Yaskawa INFORM job: vendrediTRJ2.JBI

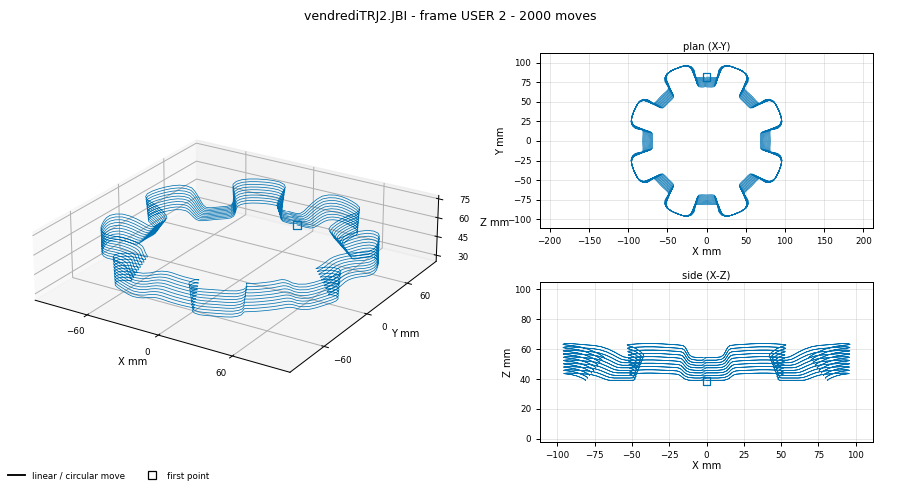
[picture p0: tool path of vendrediTRJ2.JBI in frame USER 2, 2000 of 2000 moves have a stored position in this frame; points joined in program order, loops and branches not executed]
/JOB
//NAME temp/vendrediTRJ2
///FOLDERNAME DEMO
//POS
///NPOS 2000,0,2000,0,0,0
///USER 2
///TOOL 7
///POSTYPE USER
///RECTAN
///RCONF 1,0,0,0,0,0,0,0,0,0,0,0,0,0,0,0,0,0,0,0,0,0,0,0
C00000=0.000,81.307,38.958,180.0000,38.2428,-7290.0000
C00001=4.084,81.202,38.949,-179.8245,38.2510,-7292.8792
C00002=8.115,80.931,38.962,177.3778,38.0004,-7295.7259
C00003=12.050,80.963,39.253,165.4097,32.4399,-7298.4654
C00004=14.402,82.041,39.987,165.7021,8.6017,-7299.9566
C00005=15.932,84.113,41.004,175.9998,1.1820,-7300.7254
C00006=17.234,86.943,42.060,-178.2328,-0.3684,-7301.2119
C00007=18.580,90.119,42.880,-175.4141,-1.1362,-7301.6495
C00008=20.259,92.987,43.289,-175.9026,-2.4170,-7302.2909
C00009=23.317,94.913,43.506,-178.5099,-2.2669,-7303.8024
C00010=27.389,95.566,43.684,-179.5720,-1.5763,-7305.9922
C00011=31.762,94.755,43.864,-179.9981,-0.0779,-7308.5312
C00012=36.110,93.244,43.984,179.9988,-0.0128,-7311.1696
C00013=40.400,91.468,43.984,179.9994,-0.0128,-7313.8303
C00014=44.543,89.461,43.864,179.9999,-0.0769,-7316.4689
C00015=48.209,86.942,43.684,179.5695,-1.5754,-7319.0082
C00016=50.626,83.601,43.506,178.5085,-2.2635,-7321.1977
C00017=51.426,80.077,43.289,175.9070,-2.4130,-7322.7089
C00018=50.586,76.861,42.880,175.4171,-1.1367,-7323.3509
C00019=49.291,73.664,42.060,178.2332,-0.3687,-7323.7878
C00020=48.211,70.742,41.004,-176.0002,1.1799,-7324.2746
C00021=47.828,68.195,39.987,-165.7028,8.5989,-7325.0436
C00022=48.729,65.770,39.253,-165.4121,32.4425,-7326.5348
C00023=51.488,62.965,38.962,-177.3793,38.0014,-7329.2737
C00024=54.531,60.307,38.949,179.8287,38.2519,-7332.1206
C00025=57.493,57.493,38.958,-180.0000,38.2429,-7335.0000
C00026=60.306,54.531,38.949,-179.8283,38.2519,-7337.8789
C00027=62.965,51.488,38.962,177.3793,38.0014,-7340.7263
C00028=65.770,48.729,39.253,165.4121,32.4425,-7343.4652
C00029=68.195,47.828,39.987,165.7028,8.5989,-7344.9564
C00030=70.742,48.211,41.004,176.0002,1.1799,-7345.7254
C00031=73.664,49.291,42.060,-178.2332,-0.3687,-7346.2122
C00032=76.861,50.586,42.880,-175.4171,-1.1367,-7346.6491
C00033=80.077,51.426,43.289,-175.9070,-2.4130,-7347.2911
C00034=83.601,50.626,43.506,-178.5085,-2.2635,-7348.8023
C00035=86.942,48.209,43.684,-179.5695,-1.5754,-7350.9918
C00036=89.461,44.543,43.864,-179.9999,-0.0769,-7353.5311
C00037=91.468,40.400,43.984,-179.9994,-0.0128,-7356.1697
C00038=93.244,36.110,43.984,-179.9988,-0.0128,-7358.8304
C00039=94.755,31.762,43.864,179.9981,-0.0779,-7361.4688
C00040=95.566,27.389,43.684,179.5720,-1.5763,-7364.0078
C00041=94.913,23.317,43.506,178.5099,-2.2669,-7366.1976
C00042=92.987,20.259,43.289,175.9026,-2.4170,-7367.7091
C00043=90.119,18.580,42.880,175.4141,-1.1362,-7368.3505
C00044=86.943,17.234,42.060,178.2328,-0.3684,-7368.7881
C00045=84.113,15.932,41.004,-175.9998,1.1820,-7369.2746
C00046=82.041,14.402,39.987,-165.7021,8.6017,-7370.0434
C00047=80.963,12.050,39.253,-165.4097,32.4399,-7371.5346
C00048=80.931,8.115,38.962,-177.3778,38.0004,-7374.2741
C00049=81.202,4.084,38.949,179.8245,38.2510,-7377.1208
C00050=81.307,0.000,38.958,-180.0000,38.2428,-7380.0000
C00051=81.202,-4.084,38.949,-179.8245,38.2510,-7382.8792
C00052=80.931,-8.116,38.962,177.3773,38.0004,-7385.7266
C00053=80.963,-12.050,39.253,165.4097,32.4399,-7388.4654
C00054=82.041,-14.402,39.987,165.7021,8.6017,-7389.9566
C00055=84.113,-15.932,41.004,175.9998,1.1820,-7390.7254
C00056=86.943,-17.234,42.060,-178.2328,-0.3684,-7391.2119
C00057=90.119,-18.580,42.880,-175.4141,-1.1362,-7391.6495
C00058=92.987,-20.259,43.289,-175.9026,-2.4170,-7392.2909
C00059=94.913,-23.317,43.506,-178.5099,-2.2669,-7393.8024
C00060=95.566,-27.389,43.684,-179.5720,-1.5763,-7395.9922
C00061=94.755,-31.762,43.864,-179.9981,-0.0779,-7398.5312
C00062=93.244,-36.110,43.984,179.9988,-0.0128,-7401.1696
C00063=91.468,-40.400,43.984,179.9994,-0.0128,-7403.8303
C00064=89.461,-44.543,43.864,179.9999,-0.0769,-7406.4689
C00065=86.942,-48.209,43.684,179.5695,-1.5754,-7409.0082
C00066=83.601,-50.626,43.506,178.5085,-2.2635,-7411.1977
C00067=80.077,-51.426,43.289,175.9070,-2.4130,-7412.7089
C00068=76.861,-50.586,42.880,175.4171,-1.1367,-7413.3509
C00069=73.664,-49.291,42.060,178.2332,-0.3687,-7413.7878
C00070=70.742,-48.211,41.004,-176.0002,1.1799,-7414.2746
C00071=68.195,-47.828,39.987,-165.7028,8.5989,-7415.0436
C00072=65.770,-48.729,39.253,-165.4121,32.4425,-7416.5348
C00073=62.965,-51.488,38.962,-177.3793,38.0014,-7419.2737
C00074=60.307,-54.531,38.949,179.8287,38.2519,-7422.1206
C00075=57.493,-57.493,38.958,180.0000,38.2429,-7425.0000
C00076=54.531,-60.306,38.949,-179.8283,38.2519,-7427.8789
C00077=51.488,-62.965,38.962,177.3793,38.0014,-7430.7263
C00078=48.729,-65.770,39.253,165.4121,32.4425,-7433.4652
C00079=47.828,-68.195,39.987,165.7028,8.5989,-7434.9564
C00080=48.211,-70.742,41.004,176.0002,1.1799,-7435.7254
C00081=49.291,-73.664,42.060,-178.2332,-0.3687,-7436.2122
C00082=50.586,-76.861,42.880,-175.4171,-1.1367,-7436.6491
C00083=51.426,-80.077,43.289,-175.9070,-2.4130,-7437.2911
C00084=50.626,-83.601,43.506,-178.5085,-2.2635,-7438.8023
C00085=48.209,-86.942,43.684,-179.5695,-1.5754,-7440.9918
C00086=44.543,-89.461,43.864,-179.9999,-0.0769,-7443.5311
C00087=40.400,-91.468,43.984,-179.9994,-0.0128,-7446.1697
C00088=36.110,-93.244,43.984,-179.9988,-0.0128,-7448.8304
C00089=31.762,-94.755,43.864,179.9981,-0.0779,-7451.4688
C00090=27.389,-95.566,43.684,179.5720,-1.5763,-7454.0078
C00091=23.317,-94.913,43.506,178.5099,-2.2669,-7456.1976
C00092=20.259,-92.987,43.289,175.9026,-2.4170,-7457.7091
C00093=18.580,-90.119,42.880,175.4141,-1.1362,-7458.3505
C00094=17.234,-86.943,42.060,178.2328,-0.3684,-7458.7881
C00095=15.932,-84.113,41.004,-175.9998,1.1820,-7459.2746
C00096=14.402,-82.041,39.987,-165.7021,8.6017,-7460.0434
C00097=12.050,-80.963,39.253,-165.4097,32.4399,-7461.5346
C00098=8.115,-80.931,38.962,-177.3778,38.0004,-7464.2741
C00099=4.084,-81.202,38.949,179.8245,38.2510,-7467.1208
C00100=0.000,-81.307,38.958,180.0000,38.2428,-7470.0000
C00101=-4.084,-81.202,38.949,-179.8245,38.2510,-7472.8792
C00102=-8.116,-80.931,38.962,177.3773,38.0004,-7475.7266
C00103=-12.050,-80.963,39.253,165.4097,32.4399,-7478.4654
C00104=-14.402,-82.041,39.987,165.7021,8.6017,-7479.9566
C00105=-15.932,-84.113,41.004,175.9998,1.1820,-7480.7254
C00106=-17.234,-86.943,42.060,-178.2328,-0.3684,-7481.2119
C00107=-18.580,-90.119,42.880,-175.4141,-1.1362,-7481.6495
C00108=-20.259,-92.987,43.289,-175.9026,-2.4170,-7482.2909
C00109=-23.317,-94.913,43.506,-178.5099,-2.2669,-7483.8024
C00110=-27.389,-95.566,43.684,-179.5720,-1.5763,-7485.9922
C00111=-31.762,-94.755,43.864,-179.9981,-0.0779,-7488.5312
C00112=-36.110,-93.244,43.984,179.9988,-0.0128,-7491.1696
C00113=-40.400,-91.468,43.984,179.9994,-0.0128,-7493.8303
C00114=-44.543,-89.461,43.864,179.9999,-0.0769,-7496.4689
C00115=-48.209,-86.942,43.684,179.5695,-1.5754,-7499.0082
C00116=-50.626,-83.601,43.506,178.5085,-2.2635,-7501.1977
C00117=-51.426,-80.077,43.289,175.9070,-2.4130,-7502.7089
C00118=-50.586,-76.861,42.880,175.4171,-1.1367,-7503.3509
C00119=-49.291,-73.664,42.060,178.2332,-0.3687,-7503.7878
C00120=-48.211,-70.742,41.004,-176.0002,1.1799,-7504.2746
C00121=-47.828,-68.195,39.987,-165.7028,8.5989,-7505.0436
C00122=-48.729,-65.770,39.253,-165.4121,32.4425,-7506.5348
C00123=-51.488,-62.965,38.962,-177.3793,38.0014,-7509.2737
C00124=-54.531,-60.307,38.949,179.8287,38.2519,-7512.1206
C00125=-57.493,-57.493,38.958,180.0000,38.2429,-7515.0000
C00126=-60.306,-54.531,38.949,-179.8283,38.2519,-7517.8789
C00127=-62.965,-51.488,38.962,177.3793,38.0014,-7520.7263
C00128=-65.770,-48.729,39.253,165.4121,32.4425,-7523.4652
C00129=-68.195,-47.828,39.987,165.7028,8.5989,-7524.9564
C00130=-70.742,-48.211,41.004,176.0002,1.1799,-7525.7254
C00131=-73.664,-49.291,42.060,-178.2332,-0.3687,-7526.2122
C00132=-76.861,-50.586,42.880,-175.4171,-1.1367,-7526.6491
C00133=-80.077,-51.426,43.289,-175.9070,-2.4130,-7527.2911
C00134=-83.601,-50.626,43.506,-178.5085,-2.2635,-7528.8023
C00135=-86.942,-48.209,43.684,-179.5695,-1.5754,-7530.9918
C00136=-89.461,-44.543,43.864,-179.9999,-0.0769,-7533.5311
C00137=-91.468,-40.400,43.984,-179.9994,-0.0128,-7536.1697
C00138=-93.244,-36.110,43.984,-179.9988,-0.0128,-7538.8304
C00139=-94.755,-31.762,43.864,179.9981,-0.0779,-7541.4688
C00140=-95.566,-27.389,43.684,179.5720,-1.5763,-7544.0078
C00141=-94.913,-23.317,43.506,178.5099,-2.2669,-7546.1976
C00142=-92.987,-20.259,43.289,175.9026,-2.4170,-7547.7091
C00143=-90.119,-18.580,42.880,175.4141,-1.1362,-7548.3505
C00144=-86.943,-17.234,42.060,178.2328,-0.3684,-7548.7881
C00145=-84.113,-15.932,41.004,-175.9998,1.1820,-7549.2746
C00146=-82.041,-14.402,39.987,-165.7021,8.6017,-7550.0434
C00147=-80.963,-12.050,39.253,-165.4097,32.4399,-7551.5346
C00148=-80.931,-8.115,38.962,-177.3778,38.0004,-7554.2741
C00149=-81.202,-4.084,38.949,179.8245,38.2510,-7557.1208
C00150=-81.307,0.000,38.958,180.0000,38.2428,-7560.0000
C00151=-81.202,4.084,38.949,-179.8245,38.2510,-7562.8792
C00152=-80.931,8.116,38.962,177.3773,38.0004,-7565.7266
C00153=-80.963,12.050,39.253,165.4097,32.4399,-7568.4654
C00154=-82.041,14.402,39.987,165.7021,8.6017,-7569.9566
C00155=-84.113,15.932,41.004,175.9998,1.1820,-7570.7254
C00156=-86.943,17.234,42.060,-178.2328,-0.3684,-7571.2119
C00157=-90.119,18.580,42.880,-175.4141,-1.1362,-7571.6495
C00158=-92.987,20.259,43.289,-175.9026,-2.4170,-7572.2909
C00159=-94.913,23.317,43.506,-178.5099,-2.2669,-7573.8024
C00160=-95.566,27.389,43.684,-179.5720,-1.5763,-7575.9922
C00161=-94.755,31.762,43.864,-179.9981,-0.0779,-7578.5312
C00162=-93.244,36.110,43.984,179.9988,-0.0128,-7581.1696
C00163=-91.468,40.400,43.984,179.9994,-0.0128,-7583.8303
C00164=-89.461,44.543,43.864,179.9999,-0.0769,-7586.4689
C00165=-86.942,48.209,43.684,179.5695,-1.5754,-7589.0082
C00166=-83.601,50.626,43.506,178.5085,-2.2635,-7591.1977
C00167=-80.077,51.426,43.289,175.9070,-2.4130,-7592.7089
C00168=-76.861,50.586,42.880,175.4171,-1.1367,-7593.3509
C00169=-73.664,49.291,42.060,178.2332,-0.3687,-7593.7878
C00170=-70.742,48.211,41.004,-176.0002,1.1799,-7594.2746
C00171=-68.195,47.828,39.987,-165.7028,8.5989,-7595.0436
C00172=-65.770,48.729,39.253,-165.4121,32.4425,-7596.5348
C00173=-62.965,51.488,38.962,-177.3793,38.0014,-7599.2737
C00174=-60.307,54.531,38.949,179.8287,38.2519,-7602.1206
C00175=-57.493,57.493,38.958,-180.0000,38.2429,-7605.0000
C00176=-54.531,60.306,38.949,-179.8283,38.2519,-7607.8789
C00177=-51.488,62.965,38.962,177.3793,38.0014,-7610.7263
C00178=-48.729,65.770,39.253,165.4121,32.4425,-7613.4652
C00179=-47.828,68.195,39.987,165.7028,8.5989,-7614.9564
C00180=-48.211,70.742,41.004,176.0002,1.1799,-7615.7254
C00181=-49.291,73.664,42.060,-178.2332,-0.3687,-7616.2122
C00182=-50.586,76.861,42.880,-175.4171,-1.1367,-7616.6491
C00183=-51.426,80.077,43.289,-175.9070,-2.4130,-7617.2911
C00184=-50.626,83.601,43.506,-178.5085,-2.2635,-7618.8023
C00185=-48.209,86.942,43.684,-179.5695,-1.5754,-7620.9918
C00186=-44.543,89.461,43.864,-179.9999,-0.0769,-7623.5311
C00187=-40.400,91.468,43.984,-179.9994,-0.0128,-7626.1697
C00188=-36.110,93.244,43.984,-179.9988,-0.0128,-7628.8304
C00189=-31.762,94.755,43.864,179.9981,-0.0779,-7631.4688
C00190=-27.389,95.566,43.684,179.5720,-1.5763,-7634.0078
C00191=-23.317,94.913,43.506,178.5099,-2.2669,-7636.1976
C00192=-20.259,92.987,43.289,175.9026,-2.4170,-7637.7091
C00193=-18.580,90.119,42.880,175.4141,-1.1362,-7638.3505
C00194=-17.234,86.943,42.060,178.2328,-0.3684,-7638.7881
C00195=-15.932,84.113,41.004,-175.9998,1.1820,-7639.2746
C00196=-14.402,82.041,39.987,-165.7021,8.6017,-7640.0434
C00197=-12.050,80.963,39.253,-165.4097,32.4399,-7641.5346
C00198=-8.116,80.931,38.962,-177.3773,38.0004,-7644.2734
C00199=-4.084,81.202,38.949,179.8245,38.2510,-7647.1208
C00200=0.000,79.940,40.681,-180.0000,38.6061,-7650.0000
C00201=3.959,79.840,40.672,-179.8097,38.6175,-7652.8388
C00202=7.905,79.580,40.686,177.1105,38.3368,-7655.6728
C00203=11.791,79.654,41.003,164.3962,32.0169,-7658.4202
C00204=14.083,80.839,41.802,166.7589,7.0272,-7659.8823
C00205=15.561,83.082,42.912,177.1152,0.7374,-7660.6084
C00206=16.825,86.143,44.068,-177.4031,-0.4684,-7661.0516
C00207=18.134,89.588,44.968,-174.6660,-1.1309,-7661.4429
C00208=19.771,92.721,45.418,-175.1605,-2.5717,-7662.0370
C00209=22.856,94.857,45.657,-178.2007,-2.5689,-7663.5473
C00210=27.022,95.633,45.852,-179.5051,-1.7301,-7665.7781
C00211=31.529,94.831,46.051,-179.9983,-0.0960,-7668.3907
C00212=36.031,93.275,46.182,179.9988,-0.0128,-7671.1209
C00213=40.478,91.433,46.182,179.9994,-0.0128,-7673.8793
C00214=44.762,89.350,46.051,179.9975,-0.0974,-7676.6097
C00215=48.515,86.730,45.852,179.5028,-1.7292,-7679.2218
C00216=50.913,83.236,45.657,178.2009,-2.5655,-7681.4529
C00217=51.583,79.544,45.418,175.1605,-2.5678,-7682.9628
C00218=50.526,76.172,44.968,174.6669,-1.1304,-7683.5569
C00219=49.015,72.810,44.068,177.4028,-0.4635,-7683.9481
C00220=47.744,69.752,42.912,-177.1153,0.7386,-7684.3909
C00221=47.203,67.120,41.802,-166.7608,7.0239,-7685.1173
C00222=47.986,64.662,41.003,-164.3969,32.0179,-7686.5793
C00223=50.682,61.862,40.686,-177.1071,38.3333,-7689.3269
C00224=53.655,59.255,40.672,179.8091,38.6195,-7692.1606
C00225=56.526,56.526,40.681,-180.0000,38.6039,-7695.0000
C00226=59.255,53.656,40.672,-179.8087,38.6195,-7697.8388
C00227=61.862,50.682,40.686,177.1071,38.3333,-7700.6731
C00228=64.662,47.986,41.003,164.3969,32.0179,-7703.4207
C00229=67.120,47.203,41.802,166.7608,7.0239,-7704.8827
C00230=69.752,47.744,42.912,177.1153,0.7386,-7705.6091
C00231=72.810,49.015,44.068,-177.4028,-0.4635,-7706.0519
C00232=76.172,50.526,44.968,-174.6669,-1.1304,-7706.4431
C00233=79.544,51.583,45.418,-175.1605,-2.5678,-7707.0372
C00234=83.236,50.913,45.657,-178.2009,-2.5655,-7708.5471
C00235=86.730,48.515,45.852,-179.5028,-1.7292,-7710.7782
C00236=89.350,44.762,46.051,-179.9975,-0.0974,-7713.3903
C00237=91.433,40.478,46.182,-179.9994,-0.0128,-7716.1207
C00238=93.275,36.031,46.182,-179.9988,-0.0128,-7718.8791
C00239=94.831,31.529,46.051,179.9983,-0.0960,-7721.6093
C00240=95.633,27.022,45.852,179.5051,-1.7301,-7724.2219
C00241=94.857,22.856,45.657,178.2007,-2.5689,-7726.4527
C00242=92.721,19.771,45.418,175.1605,-2.5717,-7727.9630
C00243=89.588,18.134,44.968,174.6660,-1.1309,-7728.5571
C00244=86.143,16.825,44.068,177.4031,-0.4684,-7728.9484
C00245=83.082,15.561,42.912,-177.1152,0.7374,-7729.3916
C00246=80.839,14.083,41.802,-166.7589,7.0272,-7730.1177
C00247=79.654,11.791,41.003,-164.3962,32.0169,-7731.5798
C00248=79.580,7.905,40.686,-177.1105,38.3368,-7734.3272
C00249=79.840,3.959,40.672,179.8097,38.6175,-7737.1612
C00250=79.940,0.000,40.681,-180.0000,38.6061,-7740.0000
C00251=79.840,-3.959,40.672,-179.8097,38.6175,-7742.8388
C00252=79.580,-7.905,40.686,177.1112,38.3323,-7745.6728
C00253=79.654,-11.792,41.003,164.3958,32.0168,-7748.4209
C00254=80.839,-14.083,41.802,166.7589,7.0272,-7749.8823
C00255=83.082,-15.561,42.912,177.1152,0.7374,-7750.6084
C00256=86.143,-16.825,44.068,-177.4031,-0.4684,-7751.0516
C00257=89.588,-18.134,44.968,-174.6660,-1.1309,-7751.4429
C00258=92.721,-19.771,45.418,-175.1605,-2.5717,-7752.0370
C00259=94.857,-22.856,45.657,-178.2007,-2.5689,-7753.5473
C00260=95.633,-27.022,45.852,-179.5051,-1.7301,-7755.7781
C00261=94.831,-31.529,46.051,-179.9983,-0.0960,-7758.3907
C00262=93.275,-36.031,46.182,179.9988,-0.0128,-7761.1209
C00263=91.433,-40.478,46.182,179.9994,-0.0128,-7763.8793
C00264=89.350,-44.762,46.051,179.9975,-0.0974,-7766.6097
C00265=86.730,-48.515,45.852,179.5028,-1.7292,-7769.2218
C00266=83.236,-50.913,45.657,178.2009,-2.5655,-7771.4529
C00267=79.544,-51.583,45.418,175.1605,-2.5678,-7772.9628
C00268=76.172,-50.526,44.968,174.6669,-1.1304,-7773.5569
C00269=72.810,-49.015,44.068,177.4028,-0.4635,-7773.9481
C00270=69.752,-47.744,42.912,-177.1153,0.7386,-7774.3909
C00271=67.120,-47.203,41.802,-166.7608,7.0239,-7775.1173
C00272=64.662,-47.986,41.003,-164.3969,32.0179,-7776.5793
C00273=61.862,-50.682,40.686,-177.1071,38.3333,-7779.3269
C00274=59.255,-53.655,40.672,179.8091,38.6195,-7782.1606
C00275=56.526,-56.526,40.681,-180.0000,38.6039,-7785.0000
C00276=53.656,-59.255,40.672,-179.8087,38.6195,-7787.8388
C00277=50.682,-61.862,40.686,177.1071,38.3333,-7790.6731
C00278=47.986,-64.662,41.003,164.3969,32.0179,-7793.4207
C00279=47.203,-67.120,41.802,166.7608,7.0239,-7794.8827
C00280=47.744,-69.752,42.912,177.1153,0.7386,-7795.6091
C00281=49.015,-72.810,44.068,-177.4028,-0.4635,-7796.0519
C00282=50.526,-76.172,44.968,-174.6669,-1.1304,-7796.4431
C00283=51.583,-79.544,45.418,-175.1605,-2.5678,-7797.0372
C00284=50.913,-83.236,45.657,-178.2009,-2.5655,-7798.5471
C00285=48.515,-86.730,45.852,-179.5028,-1.7292,-7800.7782
C00286=44.762,-89.350,46.051,-179.9975,-0.0974,-7803.3903
C00287=40.478,-91.433,46.182,-179.9994,-0.0128,-7806.1207
C00288=36.031,-93.275,46.182,-179.9988,-0.0128,-7808.8791
C00289=31.529,-94.831,46.051,179.9983,-0.0960,-7811.6093
C00290=27.022,-95.633,45.852,179.5051,-1.7301,-7814.2219
C00291=22.856,-94.857,45.657,178.2007,-2.5689,-7816.4527
C00292=19.771,-92.721,45.418,175.1605,-2.5717,-7817.9630
C00293=18.134,-89.588,44.968,174.6660,-1.1309,-7818.5571
C00294=16.825,-86.143,44.068,177.4031,-0.4684,-7818.9484
C00295=15.561,-83.082,42.912,-177.1152,0.7374,-7819.3916
C00296=14.083,-80.839,41.802,-166.7589,7.0272,-7820.1177
C00297=11.791,-79.654,41.003,-164.3962,32.0169,-7821.5798
C00298=7.905,-79.580,40.686,-177.1105,38.3368,-7824.3272
C00299=3.959,-79.840,40.672,179.8097,38.6175,-7827.1612
C00300=0.000,-79.940,40.681,-180.0000,38.6061,-7830.0000
C00301=-3.959,-79.840,40.672,-179.8097,38.6175,-7832.8388
C00302=-7.905,-79.580,40.686,177.1112,38.3323,-7835.6728
C00303=-11.792,-79.654,41.003,164.3958,32.0168,-7838.4209
C00304=-14.083,-80.839,41.802,166.7589,7.0272,-7839.8823
C00305=-15.561,-83.082,42.912,177.1152,0.7374,-7840.6084
C00306=-16.825,-86.143,44.068,-177.4031,-0.4684,-7841.0516
C00307=-18.134,-89.588,44.968,-174.6660,-1.1309,-7841.4429
C00308=-19.771,-92.721,45.418,-175.1605,-2.5717,-7842.0370
C00309=-22.856,-94.857,45.657,-178.2007,-2.5689,-7843.5473
C00310=-27.022,-95.633,45.852,-179.5051,-1.7301,-7845.7781
C00311=-31.529,-94.831,46.051,-179.9983,-0.0960,-7848.3907
C00312=-36.031,-93.275,46.182,179.9988,-0.0128,-7851.1209
C00313=-40.478,-91.433,46.182,179.9994,-0.0128,-7853.8793
C00314=-44.762,-89.350,46.051,179.9975,-0.0974,-7856.6097
C00315=-48.515,-86.730,45.852,179.5028,-1.7292,-7859.2218
C00316=-50.913,-83.236,45.657,178.2009,-2.5655,-7861.4529
C00317=-51.583,-79.544,45.418,175.1605,-2.5678,-7862.9628
C00318=-50.526,-76.172,44.968,174.6669,-1.1304,-7863.5569
C00319=-49.015,-72.810,44.068,177.4028,-0.4635,-7863.9481
C00320=-47.744,-69.752,42.912,-177.1153,0.7386,-7864.3909
C00321=-47.203,-67.120,41.802,-166.7608,7.0239,-7865.1173
C00322=-47.986,-64.662,41.003,-164.3969,32.0179,-7866.5793
C00323=-50.682,-61.862,40.686,-177.1071,38.3333,-7869.3269
C00324=-53.655,-59.255,40.672,179.8091,38.6195,-7872.1606
C00325=-56.526,-56.526,40.681,180.0000,38.6039,-7875.0000
C00326=-59.255,-53.656,40.672,-179.8087,38.6195,-7877.8388
C00327=-61.862,-50.682,40.686,177.1071,38.3333,-7880.6731
C00328=-64.662,-47.986,41.003,164.3969,32.0179,-7883.4207
C00329=-67.120,-47.203,41.802,166.7608,7.0239,-7884.8827
C00330=-69.752,-47.744,42.912,177.1153,0.7386,-7885.6091
C00331=-72.810,-49.015,44.068,-177.4028,-0.4635,-7886.0519
C00332=-76.172,-50.526,44.968,-174.6669,-1.1304,-7886.4431
C00333=-79.544,-51.583,45.418,-175.1605,-2.5678,-7887.0372
C00334=-83.236,-50.913,45.657,-178.2009,-2.5655,-7888.5471
C00335=-86.730,-48.515,45.852,-179.5028,-1.7292,-7890.7782
C00336=-89.350,-44.762,46.051,-179.9975,-0.0974,-7893.3903
C00337=-91.433,-40.478,46.182,-179.9994,-0.0128,-7896.1207
C00338=-93.275,-36.031,46.182,-179.9988,-0.0128,-7898.8791
C00339=-94.831,-31.529,46.051,179.9983,-0.0960,-7901.6093
C00340=-95.633,-27.022,45.852,179.5051,-1.7301,-7904.2219
C00341=-94.857,-22.856,45.657,178.2007,-2.5689,-7906.4527
C00342=-92.721,-19.771,45.418,175.1605,-2.5717,-7907.9630
C00343=-89.588,-18.134,44.968,174.6660,-1.1309,-7908.5571
C00344=-86.143,-16.825,44.068,177.4031,-0.4684,-7908.9484
C00345=-83.082,-15.561,42.912,-177.1152,0.7374,-7909.3916
C00346=-80.839,-14.083,41.802,-166.7589,7.0272,-7910.1177
C00347=-79.654,-11.791,41.003,-164.3962,32.0169,-7911.5798
C00348=-79.580,-7.905,40.686,-177.1105,38.3368,-7914.3272
C00349=-79.840,-3.959,40.672,179.8097,38.6175,-7917.1612
C00350=-79.940,0.000,40.681,180.0000,38.6061,-7920.0000
C00351=-79.840,3.959,40.672,-179.8097,38.6175,-7922.8388
C00352=-79.580,7.905,40.686,177.1112,38.3323,-7925.6728
C00353=-79.654,11.792,41.003,164.3958,32.0168,-7928.4209
C00354=-80.839,14.083,41.802,166.7589,7.0272,-7929.8823
C00355=-83.082,15.561,42.912,177.1152,0.7374,-7930.6084
C00356=-86.143,16.825,44.068,-177.4031,-0.4684,-7931.0516
C00357=-89.588,18.134,44.968,-174.6660,-1.1309,-7931.4429
C00358=-92.721,19.771,45.418,-175.1605,-2.5717,-7932.0370
C00359=-94.857,22.856,45.657,-178.2007,-2.5689,-7933.5473
C00360=-95.633,27.022,45.852,-179.5051,-1.7301,-7935.7781
C00361=-94.831,31.529,46.051,-179.9983,-0.0960,-7938.3907
C00362=-93.275,36.031,46.182,179.9988,-0.0128,-7941.1209
C00363=-91.433,40.478,46.182,179.9994,-0.0128,-7943.8793
C00364=-89.350,44.762,46.051,179.9975,-0.0974,-7946.6097
C00365=-86.730,48.515,45.852,179.5028,-1.7292,-7949.2218
C00366=-83.236,50.913,45.657,178.2009,-2.5655,-7951.4529
C00367=-79.544,51.583,45.418,175.1605,-2.5678,-7952.9628
C00368=-76.172,50.526,44.968,174.6669,-1.1304,-7953.5569
C00369=-72.810,49.015,44.068,177.4028,-0.4635,-7953.9481
C00370=-69.752,47.744,42.912,-177.1153,0.7386,-7954.3909
C00371=-67.120,47.203,41.802,-166.7608,7.0239,-7955.1173
C00372=-64.662,47.986,41.003,-164.3969,32.0179,-7956.5793
C00373=-61.862,50.682,40.686,-177.1071,38.3333,-7959.3269
C00374=-59.255,53.655,40.672,179.8091,38.6195,-7962.1606
C00375=-56.526,56.526,40.681,180.0000,38.6039,-7965.0000
C00376=-53.656,59.255,40.672,-179.8087,38.6195,-7967.8388
C00377=-50.682,61.862,40.686,177.1071,38.3333,-7970.6731
C00378=-47.986,64.662,41.003,164.3969,32.0179,-7973.4207
C00379=-47.203,67.120,41.802,166.7608,7.0239,-7974.8827
C00380=-47.744,69.752,42.912,177.1153,0.7386,-7975.6091
C00381=-49.015,72.810,44.068,-177.4028,-0.4635,-7976.0519
C00382=-50.526,76.172,44.968,-174.6669,-1.1304,-7976.4431
C00383=-51.583,79.544,45.418,-175.1605,-2.5678,-7977.0372
C00384=-50.913,83.236,45.657,-178.2009,-2.5655,-7978.5471
C00385=-48.515,86.730,45.852,-179.5028,-1.7292,-7980.7782
C00386=-44.762,89.350,46.051,-179.9975,-0.0974,-7983.3903
C00387=-40.478,91.433,46.182,-179.9994,-0.0128,-7986.1207
C00388=-36.031,93.275,46.182,-179.9988,-0.0128,-7988.8791
C00389=-31.529,94.831,46.051,179.9983,-0.0960,-7991.6093
C00390=-27.022,95.633,45.852,179.5051,-1.7301,-7994.2219
C00391=-22.856,94.857,45.657,178.2007,-2.5689,-7996.4527
C00392=-19.771,92.721,45.418,175.1605,-2.5717,-7997.9630
C00393=-18.134,89.588,44.968,174.6660,-1.1309,-7998.5571
C00394=-16.825,86.143,44.068,177.4031,-0.4684,-7998.9484
C00395=-15.561,83.082,42.912,-177.1152,0.7374,-7999.3916
C00396=-14.083,80.839,41.802,-166.7589,7.0272,-8000.1177
C00397=-11.792,79.654,41.003,-164.3958,32.0168,-8001.5791
C00398=-7.905,79.580,40.686,-177.1112,38.3323,-8004.3272
C00399=-3.959,79.840,40.672,179.8097,38.6175,-8007.1612
C00400=0.000,78.562,42.397,180.0000,38.8871,-8010.0000
C00401=3.833,78.467,42.387,-179.7965,38.9024,-8012.7966
C00402=7.694,78.220,42.402,176.8336,38.5856,-8015.6177
C00403=11.532,78.336,42.745,163.4668,31.4523,-8018.3745
C00404=13.762,79.628,43.611,167.9418,5.6496,-8019.8055
C00405=15.189,82.045,44.816,178.1581,0.4109,-8020.4884
C00406=16.414,85.339,46.074,-176.6678,-0.5097,-8020.8872
C00407=17.687,89.056,47.055,-174.0207,-1.0814,-8021.2331
C00408=19.281,92.454,47.546,-174.4848,-2.6470,-8021.7800
C00409=22.392,94.802,47.807,-177.8991,-2.8280,-8023.2896
C00410=26.654,95.700,48.020,-179.4439,-1.8679,-8025.5634
C00411=31.296,94.909,48.237,179.9996,-0.1087,-8028.2498
C00412=35.952,93.306,48.381,179.9988,-0.0128,-8031.0723
C00413=40.555,91.399,48.381,179.9994,-0.0128,-8033.9275
C00414=44.981,89.240,48.237,179.9978,-0.1102,-8036.7502
C00415=48.823,86.517,48.020,179.4417,-1.8680,-8039.4368
C00416=51.201,82.869,47.807,177.9023,-2.8261,-8041.7100
C00417=51.741,79.009,47.546,174.4861,-2.6490,-8043.2198
C00418=50.465,75.478,47.055,174.0210,-1.0802,-8043.7669
C00419=48.737,71.950,46.074,176.6694,-0.5117,-8044.1127
C00420=47.275,68.755,44.816,-178.1605,0.4096,-8044.5119
C00421=46.575,66.037,43.611,-167.9415,5.6466,-8045.1948
C00422=47.238,63.546,42.745,-163.4715,31.4493,-8046.6259
C00423=49.870,60.750,42.402,-176.8306,38.5888,-8049.3828
C00424=52.774,58.195,42.387,179.7983,38.9007,-8052.2032
C00425=55.552,55.552,42.397,180.0000,38.8857,-8055.0000
C00426=58.195,52.774,42.387,-179.7983,38.9007,-8057.7968
C00427=60.750,49.870,42.402,176.8310,38.5853,-8060.6172
C00428=63.546,47.238,42.745,163.4715,31.4493,-8063.3741
C00429=66.037,46.575,43.611,167.9415,5.6466,-8064.8052
C00430=68.755,47.275,44.816,178.1605,0.4096,-8065.4881
C00431=71.950,48.737,46.074,-176.6694,-0.5117,-8065.8873
C00432=75.478,50.465,47.055,-174.0210,-1.0802,-8066.2331
C00433=79.009,51.741,47.546,-174.4861,-2.6490,-8066.7802
C00434=82.869,51.201,47.807,-177.9023,-2.8261,-8068.2900
C00435=86.517,48.823,48.020,-179.4417,-1.8680,-8070.5632
C00436=89.240,44.981,48.237,-179.9978,-0.1102,-8073.2498
C00437=91.399,40.555,48.381,-179.9994,-0.0128,-8076.0725
C00438=93.306,35.952,48.381,-179.9988,-0.0128,-8078.9277
C00439=94.909,31.296,48.237,-179.9996,-0.1087,-8081.7502
C00440=95.700,26.654,48.020,179.4439,-1.8679,-8084.4366
C00441=94.802,22.392,47.807,177.8991,-2.8280,-8086.7104
C00442=92.454,19.281,47.546,174.4848,-2.6470,-8088.2200
C00443=89.056,17.687,47.055,174.0207,-1.0814,-8088.7669
C00444=85.339,16.414,46.074,176.6678,-0.5097,-8089.1128
C00445=82.045,15.189,44.816,-178.1581,0.4109,-8089.5116
C00446=79.628,13.762,43.611,-167.9418,5.6496,-8090.1945
C00447=78.336,11.532,42.745,-163.4668,31.4523,-8091.6255
C00448=78.220,7.694,42.402,-176.8336,38.5856,-8094.3823
C00449=78.467,3.833,42.387,179.7965,38.9024,-8097.2034
C00450=78.562,0.000,42.397,-180.0000,38.8871,-8100.0000
C00451=78.467,-3.833,42.387,-179.7965,38.9024,-8102.7966
C00452=78.220,-7.694,42.402,176.8267,38.5816,-8105.6177
C00453=78.336,-11.532,42.745,163.4668,31.4523,-8108.3745
C00454=79.628,-13.762,43.611,167.9418,5.6496,-8109.8055
C00455=82.045,-15.189,44.816,178.1581,0.4109,-8110.4884
C00456=85.339,-16.414,46.074,-176.6678,-0.5097,-8110.8872
C00457=89.056,-17.687,47.055,-174.0207,-1.0814,-8111.2331
C00458=92.454,-19.281,47.546,-174.4848,-2.6470,-8111.7800
C00459=94.802,-22.392,47.807,-177.8991,-2.8280,-8113.2896
C00460=95.700,-26.654,48.020,-179.4439,-1.8679,-8115.5634
C00461=94.909,-31.296,48.237,179.9996,-0.1087,-8118.2498
C00462=93.306,-35.952,48.381,179.9988,-0.0128,-8121.0723
C00463=91.399,-40.555,48.381,179.9994,-0.0128,-8123.9275
C00464=89.240,-44.981,48.237,179.9978,-0.1102,-8126.7502
C00465=86.517,-48.823,48.020,179.4417,-1.8680,-8129.4368
C00466=82.869,-51.201,47.807,177.9023,-2.8261,-8131.7100
C00467=79.009,-51.741,47.546,174.4861,-2.6490,-8133.2198
C00468=75.478,-50.465,47.055,174.0210,-1.0802,-8133.7669
C00469=71.950,-48.737,46.074,176.6694,-0.5117,-8134.1127
C00470=68.755,-47.275,44.816,-178.1605,0.4096,-8134.5119
C00471=66.037,-46.575,43.611,-167.9415,5.6466,-8135.1948
C00472=63.546,-47.238,42.745,-163.4715,31.4493,-8136.6259
C00473=60.750,-49.870,42.402,-176.8306,38.5888,-8139.3828
C00474=58.195,-52.774,42.387,179.7983,38.9007,-8142.2032
C00475=55.552,-55.552,42.397,-180.0000,38.8857,-8145.0000
C00476=52.774,-58.195,42.387,-179.7983,38.9007,-8147.7968
C00477=49.870,-60.750,42.402,176.8310,38.5853,-8150.6172
C00478=47.238,-63.546,42.745,163.4715,31.4493,-8153.3741
C00479=46.575,-66.037,43.611,167.9415,5.6466,-8154.8052
C00480=47.275,-68.755,44.816,178.1605,0.4096,-8155.4881
C00481=48.737,-71.950,46.074,-176.6694,-0.5117,-8155.8873
C00482=50.465,-75.478,47.055,-174.0210,-1.0802,-8156.2331
C00483=51.741,-79.009,47.546,-174.4861,-2.6490,-8156.7802
C00484=51.201,-82.869,47.807,-177.9023,-2.8261,-8158.2900
C00485=48.823,-86.517,48.020,-179.4417,-1.8680,-8160.5632
C00486=44.981,-89.240,48.237,-179.9978,-0.1102,-8163.2498
C00487=40.555,-91.399,48.381,-179.9994,-0.0128,-8166.0725
C00488=35.952,-93.306,48.381,-179.9988,-0.0128,-8168.9277
C00489=31.296,-94.909,48.237,-179.9996,-0.1087,-8171.7502
C00490=26.654,-95.700,48.020,179.4439,-1.8679,-8174.4366
C00491=22.392,-94.802,47.807,177.8991,-2.8280,-8176.7104
C00492=19.281,-92.454,47.546,174.4848,-2.6470,-8178.2200
C00493=17.687,-89.056,47.055,174.0207,-1.0814,-8178.7669
C00494=16.414,-85.339,46.074,176.6678,-0.5097,-8179.1128
C00495=15.189,-82.045,44.816,-178.1581,0.4109,-8179.5116
C00496=13.762,-79.628,43.611,-167.9418,5.6496,-8180.1945
C00497=11.532,-78.336,42.745,-163.4668,31.4523,-8181.6255
C00498=7.694,-78.220,42.402,-176.8336,38.5856,-8184.3823
C00499=3.833,-78.467,42.387,179.7965,38.9024,-8187.2034
C00500=0.000,-78.562,42.397,-180.0000,38.8871,-8190.0000
C00501=-3.833,-78.467,42.387,-179.7965,38.9024,-8192.7966
C00502=-7.694,-78.220,42.402,176.8267,38.5816,-8195.6177
C00503=-11.532,-78.336,42.745,163.4668,31.4523,-8198.3745
C00504=-13.762,-79.628,43.611,167.9418,5.6496,-8199.8055
C00505=-15.189,-82.045,44.816,178.1581,0.4109,-8200.4884
C00506=-16.414,-85.339,46.074,-176.6678,-0.5097,-8200.8872
C00507=-17.687,-89.056,47.055,-174.0207,-1.0814,-8201.2331
C00508=-19.281,-92.454,47.546,-174.4848,-2.6470,-8201.7800
C00509=-22.392,-94.802,47.807,-177.8991,-2.8280,-8203.2896
C00510=-26.654,-95.700,48.020,-179.4439,-1.8679,-8205.5634
C00511=-31.296,-94.909,48.237,179.9996,-0.1087,-8208.2498
C00512=-35.952,-93.306,48.381,179.9988,-0.0128,-8211.0723
C00513=-40.555,-91.399,48.381,179.9994,-0.0128,-8213.9275
C00514=-44.981,-89.240,48.237,179.9978,-0.1102,-8216.7502
C00515=-48.823,-86.517,48.020,179.4417,-1.8680,-8219.4368
C00516=-51.201,-82.869,47.807,177.9023,-2.8261,-8221.7100
C00517=-51.741,-79.009,47.546,174.4861,-2.6490,-8223.2198
C00518=-50.465,-75.478,47.055,174.0210,-1.0802,-8223.7669
C00519=-48.737,-71.950,46.074,176.6694,-0.5117,-8224.1127
C00520=-47.275,-68.755,44.816,-178.1605,0.4096,-8224.5119
C00521=-46.575,-66.037,43.611,-167.9415,5.6466,-8225.1948
C00522=-47.238,-63.546,42.745,-163.4715,31.4493,-8226.6259
C00523=-49.870,-60.750,42.402,-176.8306,38.5888,-8229.3828
C00524=-52.774,-58.195,42.387,179.7983,38.9007,-8232.2032
C00525=-55.552,-55.552,42.397,-180.0000,38.8857,-8235.0000
C00526=-58.195,-52.774,42.387,-179.7983,38.9007,-8237.7968
C00527=-60.750,-49.870,42.402,176.8310,38.5853,-8240.6172
C00528=-63.546,-47.238,42.745,163.4715,31.4493,-8243.3741
C00529=-66.037,-46.575,43.611,167.9415,5.6466,-8244.8052
C00530=-68.755,-47.275,44.816,178.1605,0.4096,-8245.4881
C00531=-71.950,-48.737,46.074,-176.6694,-0.5117,-8245.8873
C00532=-75.478,-50.465,47.055,-174.0210,-1.0802,-8246.2331
C00533=-79.009,-51.741,47.546,-174.4861,-2.6490,-8246.7802
C00534=-82.869,-51.201,47.807,-177.9023,-2.8261,-8248.2900
C00535=-86.517,-48.823,48.020,-179.4417,-1.8680,-8250.5632
C00536=-89.240,-44.981,48.237,-179.9978,-0.1102,-8253.2498
C00537=-91.399,-40.555,48.381,-179.9994,-0.0128,-8256.0725
C00538=-93.306,-35.952,48.381,-179.9988,-0.0128,-8258.9277
C00539=-94.909,-31.296,48.237,-179.9996,-0.1087,-8261.7502
C00540=-95.700,-26.654,48.020,179.4439,-1.8679,-8264.4366
C00541=-94.802,-22.392,47.807,177.8991,-2.8280,-8266.7104
C00542=-92.454,-19.281,47.546,174.4848,-2.6470,-8268.2200
C00543=-89.056,-17.687,47.055,174.0207,-1.0814,-8268.7669
C00544=-85.339,-16.414,46.074,176.6678,-0.5097,-8269.1128
C00545=-82.045,-15.189,44.816,-178.1581,0.4109,-8269.5116
C00546=-79.628,-13.762,43.611,-167.9418,5.6496,-8270.1945
C00547=-78.336,-11.532,42.745,-163.4668,31.4523,-8271.6255
C00548=-78.220,-7.694,42.402,-176.8336,38.5856,-8274.3823
C00549=-78.467,-3.833,42.387,179.7965,38.9024,-8277.2034
C00550=-78.562,0.000,42.397,-180.0000,38.8871,-8280.0000
C00551=-78.467,3.833,42.387,-179.7965,38.9024,-8282.7966
C00552=-78.220,7.694,42.402,176.8267,38.5816,-8285.6177
C00553=-78.336,11.532,42.745,163.4668,31.4523,-8288.3745
C00554=-79.628,13.762,43.611,167.9418,5.6496,-8289.8055
C00555=-82.045,15.189,44.816,178.1581,0.4109,-8290.4884
C00556=-85.339,16.414,46.074,-176.6678,-0.5097,-8290.8872
C00557=-89.056,17.687,47.055,-174.0207,-1.0814,-8291.2331
C00558=-92.454,19.281,47.546,-174.4848,-2.6470,-8291.7800
C00559=-94.802,22.392,47.807,-177.8991,-2.8280,-8293.2896
C00560=-95.700,26.654,48.020,-179.4439,-1.8679,-8295.5634
C00561=-94.909,31.296,48.237,179.9996,-0.1087,-8298.2498
C00562=-93.306,35.952,48.381,179.9988,-0.0128,-8301.0723
C00563=-91.399,40.555,48.381,179.9994,-0.0128,-8303.9275
C00564=-89.240,44.981,48.237,179.9978,-0.1102,-8306.7502
C00565=-86.517,48.823,48.020,179.4417,-1.8680,-8309.4368
C00566=-82.869,51.201,47.807,177.9023,-2.8261,-8311.7100
C00567=-79.009,51.741,47.546,174.4861,-2.6490,-8313.2198
C00568=-75.478,50.465,47.055,174.0210,-1.0802,-8313.7669
C00569=-71.950,48.737,46.074,176.6694,-0.5117,-8314.1127
C00570=-68.755,47.275,44.816,-178.1605,0.4096,-8314.5119
C00571=-66.037,46.575,43.611,-167.9415,5.6466,-8315.1948
C00572=-63.546,47.238,42.745,-163.4715,31.4493,-8316.6259
C00573=-60.750,49.870,42.402,-176.8306,38.5888,-8319.3828
C00574=-58.195,52.774,42.387,179.7983,38.9007,-8322.2032
C00575=-55.552,55.552,42.397,-180.0000,38.8857,-8325.0000
C00576=-52.774,58.195,42.387,-179.7983,38.9007,-8327.7968
C00577=-49.870,60.750,42.402,176.8310,38.5853,-8330.6172
C00578=-47.238,63.546,42.745,163.4715,31.4493,-8333.3741
C00579=-46.575,66.037,43.611,167.9415,5.6466,-8334.8052
C00580=-47.275,68.755,44.816,178.1605,0.4096,-8335.4881
C00581=-48.737,71.950,46.074,-176.6694,-0.5117,-8335.8873
C00582=-50.465,75.478,47.055,-174.0210,-1.0802,-8336.2331
C00583=-51.741,79.009,47.546,-174.4861,-2.6490,-8336.7802
C00584=-51.201,82.869,47.807,-177.9023,-2.8261,-8338.2900
C00585=-48.823,86.517,48.020,-179.4417,-1.8680,-8340.5632
C00586=-44.981,89.240,48.237,-179.9978,-0.1102,-8343.2498
C00587=-40.555,91.399,48.381,-179.9994,-0.0128,-8346.0725
C00588=-35.952,93.306,48.381,-179.9988,-0.0128,-8348.9277
C00589=-31.296,94.909,48.237,-179.9996,-0.1087,-8351.7502
C00590=-26.654,95.700,48.020,179.4439,-1.8679,-8354.4366
C00591=-22.392,94.802,47.807,177.8991,-2.8280,-8356.7104
C00592=-19.281,92.454,47.546,174.4848,-2.6470,-8358.2200
C00593=-17.687,89.056,47.055,174.0207,-1.0814,-8358.7669
C00594=-16.414,85.339,46.074,176.6678,-0.5097,-8359.1128
C00595=-15.189,82.045,44.816,-178.1581,0.4109,-8359.5116
C00596=-13.762,79.628,43.611,-167.9418,5.6496,-8360.1945
C00597=-11.532,78.336,42.745,-163.4668,31.4523,-8361.6255
C00598=-7.694,78.220,42.402,-176.8267,38.5816,-8364.3823
C00599=-3.833,78.467,42.387,179.7965,38.9024,-8367.2034
C00600=0.000,77.178,44.107,180.0000,39.0947,-8370.0000
C00601=3.707,77.088,44.096,-179.7781,39.1060,-8372.7531
C00602=7.481,76.852,44.112,176.5472,38.7533,-8375.5598
C00603=11.270,77.011,44.481,162.6489,30.7477,-8378.3257
C00604=13.439,78.412,45.416,169.2009,4.4687,-8379.7254
C00605=14.814,81.004,46.718,179.1240,0.1718,-8380.3637
C00606=16.001,84.532,48.079,-176.0265,-0.5209,-8380.7187
C00607=17.239,88.522,49.141,-173.4751,-1.0036,-8381.0200
C00608=18.791,92.187,49.674,-173.8989,-2.6645,-8381.5211
C00609=21.929,94.746,49.957,-177.6156,-3.0465,-8383.0317
C00610=26.285,95.767,50.188,-179.3828,-1.9881,-8385.3479
C00611=31.062,94.986,50.423,-179.9971,-0.1196,-8388.1086
C00612=35.872,93.336,50.579,179.9988,-0.0128,-8391.0234
C00613=40.633,91.364,50.579,179.9994,-0.0128,-8393.9765
C00614=45.201,89.129,50.423,179.9955,-0.1179,-8396.8914
C00615=49.131,86.304,50.188,179.3831,-1.9866,-8399.6519
C00616=51.489,82.502,49.957,177.6168,-3.0423,-8401.9680
C00617=51.899,78.473,49.674,173.8972,-2.6664,-8403.4791
C00618=50.405,74.784,49.141,173.4748,-1.0089,-8403.9803
C00619=48.459,71.088,48.079,176.0261,-0.5237,-8404.2813
C00620=46.803,67.754,46.718,-179.1207,0.1687,-8404.6359
C00621=45.943,64.949,45.416,-169.2015,4.4679,-8405.2745
C00622=46.486,62.424,44.481,-162.6478,30.7469,-8406.6744
C00623=49.053,59.633,44.112,-176.5513,38.7545,-8409.4401
C00624=51.888,57.130,44.096,179.7827,39.1054,-8412.2471
C00625=54.573,54.573,44.107,180.0000,39.0946,-8415.0000
C00626=57.130,51.888,44.096,-179.7827,39.1054,-8417.7529
C00627=59.633,49.053,44.112,176.5513,38.7545,-8420.5599
C00628=62.424,46.486,44.482,162.6515,30.7510,-8423.3256
C00629=64.949,45.943,45.416,169.2015,4.4679,-8424.7255
C00630=67.754,46.803,46.718,179.1207,0.1687,-8425.3641
C00631=71.088,48.459,48.079,-176.0261,-0.5237,-8425.7187
C00632=74.784,50.405,49.141,-173.4748,-1.0089,-8426.0197
C00633=78.473,51.899,49.674,-173.8972,-2.6664,-8426.5209
C00634=82.502,51.489,49.957,-177.6168,-3.0423,-8428.0320
C00635=86.304,49.131,50.188,-179.3831,-1.9866,-8430.3481
C00636=89.129,45.201,50.423,-179.9955,-0.1179,-8433.1086
C00637=91.364,40.633,50.579,-179.9994,-0.0128,-8436.0235
C00638=93.336,35.872,50.579,-179.9988,-0.0128,-8438.9766
C00639=94.986,31.062,50.423,179.9971,-0.1196,-8441.8914
C00640=95.767,26.285,50.188,179.3828,-1.9881,-8444.6521
C00641=94.746,21.929,49.957,177.6156,-3.0465,-8446.9683
C00642=92.187,18.791,49.674,173.8989,-2.6645,-8448.4789
C00643=88.522,17.239,49.141,173.4751,-1.0036,-8448.9800
C00644=84.532,16.001,48.079,176.0265,-0.5209,-8449.2813
C00645=81.004,14.814,46.718,-179.1240,0.1718,-8449.6363
C00646=78.412,13.439,45.416,-169.2009,4.4687,-8450.2746
C00647=77.011,11.270,44.481,-162.6489,30.7477,-8451.6743
C00648=76.852,7.481,44.112,-176.5472,38.7533,-8454.4402
C00649=77.088,3.707,44.096,179.7781,39.1060,-8457.2469
C00650=77.178,0.000,44.107,180.0000,39.0947,-8460.0000
C00651=77.088,-3.707,44.096,-179.7781,39.1060,-8462.7531
C00652=76.852,-7.481,44.112,176.5472,38.7533,-8465.5598
C00653=77.011,-11.270,44.482,162.6489,30.7477,-8468.3257
C00654=78.412,-13.439,45.416,169.2009,4.4687,-8469.7254
C00655=81.004,-14.814,46.718,179.1240,0.1718,-8470.3637
C00656=84.532,-16.001,48.079,-176.0265,-0.5209,-8470.7187
C00657=88.522,-17.239,49.141,-173.4751,-1.0036,-8471.0200
C00658=92.187,-18.791,49.674,-173.8989,-2.6645,-8471.5211
C00659=94.746,-21.929,49.957,-177.6156,-3.0465,-8473.0317
C00660=95.767,-26.285,50.188,-179.3828,-1.9881,-8475.3479
C00661=94.986,-31.062,50.423,-179.9971,-0.1196,-8478.1086
C00662=93.336,-35.872,50.579,179.9988,-0.0128,-8481.0234
C00663=91.364,-40.633,50.579,179.9994,-0.0128,-8483.9765
C00664=89.129,-45.201,50.423,179.9955,-0.1179,-8486.8914
C00665=86.304,-49.131,50.188,179.3831,-1.9866,-8489.6519
C00666=82.502,-51.489,49.957,177.6168,-3.0423,-8491.9680
C00667=78.473,-51.899,49.674,173.8972,-2.6664,-8493.4791
C00668=74.784,-50.405,49.141,173.4748,-1.0089,-8493.9803
C00669=71.088,-48.459,48.079,176.0261,-0.5237,-8494.2813
C00670=67.754,-46.803,46.718,-179.1207,0.1687,-8494.6359
C00671=64.949,-45.943,45.416,-169.2015,4.4679,-8495.2745
C00672=62.424,-46.486,44.481,-162.6478,30.7469,-8496.6744
C00673=59.633,-49.053,44.112,-176.5513,38.7545,-8499.4401
C00674=57.130,-51.888,44.096,179.7827,39.1054,-8502.2471
C00675=54.573,-54.573,44.107,180.0000,39.0946,-8505.0000
C00676=51.888,-57.130,44.096,-179.7827,39.1054,-8507.7529
C00677=49.053,-59.633,44.112,176.5513,38.7545,-8510.5599
C00678=46.486,-62.424,44.482,162.6515,30.7510,-8513.3256
C00679=45.943,-64.949,45.416,169.2015,4.4679,-8514.7255
C00680=46.803,-67.754,46.718,179.1207,0.1687,-8515.3641
C00681=48.459,-71.088,48.079,-176.0261,-0.5237,-8515.7187
C00682=50.405,-74.784,49.141,-173.4748,-1.0089,-8516.0197
C00683=51.899,-78.473,49.674,-173.8972,-2.6664,-8516.5209
C00684=51.489,-82.502,49.957,-177.6168,-3.0423,-8518.0320
C00685=49.131,-86.304,50.188,-179.3831,-1.9866,-8520.3481
C00686=45.201,-89.129,50.423,-179.9955,-0.1179,-8523.1086
C00687=40.633,-91.364,50.579,-179.9994,-0.0128,-8526.0235
C00688=35.872,-93.336,50.579,-179.9988,-0.0128,-8528.9766
C00689=31.062,-94.986,50.423,179.9971,-0.1196,-8531.8914
C00690=26.285,-95.767,50.188,179.3828,-1.9881,-8534.6521
C00691=21.929,-94.746,49.957,177.6156,-3.0465,-8536.9683
C00692=18.791,-92.187,49.674,173.8989,-2.6645,-8538.4789
C00693=17.239,-88.522,49.141,173.4751,-1.0036,-8538.9800
C00694=16.001,-84.532,48.079,176.0265,-0.5209,-8539.2813
C00695=14.814,-81.004,46.718,-179.1240,0.1718,-8539.6363
C00696=13.439,-78.412,45.416,-169.2009,4.4687,-8540.2746
C00697=11.270,-77.011,44.481,-162.6489,30.7477,-8541.6743
C00698=7.481,-76.852,44.112,-176.5472,38.7533,-8544.4402
C00699=3.707,-77.088,44.096,179.7781,39.1060,-8547.2469
C00700=0.000,-77.178,44.107,-180.0000,39.0947,-8550.0000
C00701=-3.707,-77.088,44.096,-179.7781,39.1060,-8552.7531
C00702=-7.481,-76.852,44.112,176.5472,38.7533,-8555.5598
C00703=-11.270,-77.011,44.482,162.6489,30.7477,-8558.3257
C00704=-13.439,-78.412,45.416,169.2009,4.4687,-8559.7254
C00705=-14.814,-81.004,46.718,179.1240,0.1718,-8560.3637
C00706=-16.001,-84.532,48.079,-176.0265,-0.5209,-8560.7187
C00707=-17.239,-88.522,49.141,-173.4751,-1.0036,-8561.0200
C00708=-18.791,-92.187,49.674,-173.8989,-2.6645,-8561.5211
C00709=-21.929,-94.746,49.957,-177.6156,-3.0465,-8563.0317
C00710=-26.285,-95.767,50.188,-179.3828,-1.9881,-8565.3479
C00711=-31.062,-94.986,50.423,-179.9971,-0.1196,-8568.1086
C00712=-35.872,-93.336,50.579,179.9988,-0.0128,-8571.0234
C00713=-40.633,-91.364,50.579,179.9994,-0.0128,-8573.9765
C00714=-45.201,-89.129,50.423,179.9955,-0.1179,-8576.8914
C00715=-49.131,-86.304,50.188,179.3831,-1.9866,-8579.6519
C00716=-51.489,-82.502,49.957,177.6168,-3.0423,-8581.9680
C00717=-51.899,-78.473,49.674,173.8972,-2.6664,-8583.4791
C00718=-50.405,-74.784,49.141,173.4748,-1.0089,-8583.9803
C00719=-48.459,-71.088,48.079,176.0261,-0.5237,-8584.2813
C00720=-46.803,-67.754,46.718,-179.1207,0.1687,-8584.6359
C00721=-45.943,-64.949,45.416,-169.2015,4.4679,-8585.2745
C00722=-46.486,-62.424,44.481,-162.6478,30.7469,-8586.6744
C00723=-49.053,-59.633,44.112,-176.5513,38.7545,-8589.4401
C00724=-51.888,-57.130,44.096,179.7827,39.1054,-8592.2471
C00725=-54.573,-54.573,44.107,-180.0000,39.0946,-8595.0000
C00726=-57.130,-51.888,44.096,-179.7827,39.1054,-8597.7529
C00727=-59.633,-49.053,44.112,176.5513,38.7545,-8600.5599
C00728=-62.424,-46.486,44.482,162.6515,30.7510,-8603.3256
C00729=-64.949,-45.943,45.416,169.2015,4.4679,-8604.7255
C00730=-67.754,-46.803,46.718,179.1207,0.1687,-8605.3641
C00731=-71.088,-48.459,48.079,-176.0261,-0.5237,-8605.7187
C00732=-74.784,-50.405,49.141,-173.4748,-1.0089,-8606.0197
C00733=-78.473,-51.899,49.674,-173.8972,-2.6664,-8606.5209
C00734=-82.502,-51.489,49.957,-177.6168,-3.0423,-8608.0320
C00735=-86.304,-49.131,50.188,-179.3831,-1.9866,-8610.3481
C00736=-89.129,-45.201,50.423,-179.9955,-0.1179,-8613.1086
C00737=-91.364,-40.633,50.579,-179.9994,-0.0128,-8616.0235
C00738=-93.336,-35.872,50.579,-179.9988,-0.0128,-8618.9766
C00739=-94.986,-31.062,50.423,179.9971,-0.1196,-8621.8914
C00740=-95.767,-26.285,50.188,179.3828,-1.9881,-8624.6521
C00741=-94.746,-21.929,49.957,177.6156,-3.0465,-8626.9683
C00742=-92.187,-18.791,49.674,173.8989,-2.6645,-8628.4789
C00743=-88.522,-17.239,49.141,173.4751,-1.0036,-8628.9800
C00744=-84.532,-16.001,48.079,176.0265,-0.5209,-8629.2813
C00745=-81.004,-14.814,46.718,-179.1240,0.1718,-8629.6363
C00746=-78.412,-13.439,45.416,-169.2009,4.4687,-8630.2746
C00747=-77.011,-11.270,44.481,-162.6489,30.7477,-8631.6743
C00748=-76.852,-7.481,44.112,-176.5472,38.7533,-8634.4402
C00749=-77.088,-3.707,44.096,179.7781,39.1060,-8637.2469
C00750=-77.178,0.000,44.107,-180.0000,39.0947,-8640.0000
C00751=-77.088,3.707,44.096,-179.7781,39.1060,-8642.7531
C00752=-76.852,7.481,44.112,176.5472,38.7533,-8645.5598
C00753=-77.011,11.270,44.482,162.6489,30.7477,-8648.3257
C00754=-78.412,13.439,45.416,169.2009,4.4687,-8649.7254
C00755=-81.004,14.814,46.718,179.1240,0.1718,-8650.3637
C00756=-84.532,16.001,48.079,-176.0265,-0.5209,-8650.7187
C00757=-88.522,17.239,49.141,-173.4751,-1.0036,-8651.0200
C00758=-92.187,18.791,49.674,-173.8989,-2.6645,-8651.5211
C00759=-94.746,21.929,49.957,-177.6156,-3.0465,-8653.0317
C00760=-95.767,26.285,50.188,-179.3828,-1.9881,-8655.3479
C00761=-94.986,31.062,50.423,-179.9971,-0.1196,-8658.1086
C00762=-93.336,35.872,50.579,179.9988,-0.0128,-8661.0234
C00763=-91.364,40.633,50.579,179.9994,-0.0128,-8663.9765
C00764=-89.129,45.201,50.423,179.9955,-0.1179,-8666.8914
C00765=-86.304,49.131,50.188,179.3831,-1.9866,-8669.6519
C00766=-82.502,51.489,49.957,177.6168,-3.0423,-8671.9680
C00767=-78.473,51.899,49.674,173.8972,-2.6664,-8673.4791
C00768=-74.784,50.405,49.141,173.4748,-1.0089,-8673.9803
C00769=-71.088,48.459,48.079,176.0261,-0.5237,-8674.2813
C00770=-67.754,46.803,46.718,-179.1207,0.1687,-8674.6359
C00771=-64.949,45.943,45.416,-169.2015,4.4679,-8675.2745
C00772=-62.424,46.486,44.481,-162.6478,30.7469,-8676.6744
C00773=-59.633,49.053,44.112,-176.5513,38.7545,-8679.4401
C00774=-57.130,51.888,44.096,179.7827,39.1054,-8682.2471
C00775=-54.573,54.573,44.107,-180.0000,39.0946,-8685.0000
C00776=-51.888,57.130,44.096,-179.7827,39.1054,-8687.7529
C00777=-49.053,59.633,44.112,176.5513,38.7545,-8690.5599
C00778=-46.486,62.424,44.482,162.6515,30.7510,-8693.3256
C00779=-45.943,64.949,45.416,169.2015,4.4679,-8694.7255
C00780=-46.803,67.754,46.718,179.1207,0.1687,-8695.3641
C00781=-48.459,71.088,48.079,-176.0261,-0.5237,-8695.7187
C00782=-50.405,74.784,49.141,-173.4748,-1.0089,-8696.0197
C00783=-51.899,78.473,49.674,-173.8972,-2.6664,-8696.5209
C00784=-51.489,82.502,49.957,-177.6168,-3.0423,-8698.0320
C00785=-49.131,86.304,50.188,-179.3831,-1.9866,-8700.3481
C00786=-45.201,89.129,50.423,-179.9955,-0.1179,-8703.1086
C00787=-40.633,91.364,50.579,-179.9994,-0.0128,-8706.0235
C00788=-35.872,93.336,50.579,-179.9988,-0.0128,-8708.9766
C00789=-31.062,94.986,50.423,179.9971,-0.1196,-8711.8914
C00790=-26.285,95.767,50.188,179.3828,-1.9881,-8714.6521
C00791=-21.929,94.746,49.957,177.6156,-3.0465,-8716.9683
C00792=-18.791,92.187,49.674,173.8989,-2.6645,-8718.4789
C00793=-17.239,88.522,49.141,173.4751,-1.0036,-8718.9800
C00794=-16.001,84.532,48.079,176.0265,-0.5209,-8719.2813
C00795=-14.814,81.004,46.718,-179.1240,0.1718,-8719.6363
C00796=-13.439,78.412,45.416,-169.2009,4.4687,-8720.2746
C00797=-11.270,77.011,44.482,-162.6489,30.7477,-8721.6743
C00798=-7.481,76.852,44.112,-176.5472,38.7533,-8724.4402
C00799=-3.707,77.088,44.096,179.7781,39.1060,-8727.2469
C00800=0.000,75.789,45.812,-180.0000,39.2289,-8730.0000
C00801=3.580,75.703,45.801,-179.7689,39.2394,-8732.7075
C00802=7.267,75.480,45.818,176.2657,38.8470,-8735.4993
C00803=11.008,75.681,46.215,161.9441,29.9170,-8738.2758
C00804=13.116,77.193,47.218,170.4942,3.4778,-8739.6431
C00805=14.439,79.961,48.618,179.9944,-0.0010,-8740.2359
C00806=15.588,83.726,50.084,-175.4718,-0.5058,-8740.5465
C00807=16.791,87.989,51.229,-173.0243,-0.9189,-8740.8039
C00808=18.302,91.921,51.802,-173.3993,-2.6344,-8741.2607
C00809=21.467,94.690,52.107,-177.3556,-3.2253,-8742.7735
C00810=25.919,95.834,52.356,-179.3271,-2.0919,-8745.1340
C00811=30.830,95.062,52.610,-179.9993,-0.1323,-8747.9686
C00812=35.794,93.367,52.777,-179.9992,-0.0181,-8750.9753
C00813=40.710,91.330,52.777,-179.9982,-0.0180,-8754.0247
C00814=45.419,89.019,52.610,179.9959,-0.1307,-8757.0314
C00815=49.437,86.092,52.356,179.3324,-2.0949,-8759.8659
C00816=51.776,82.136,52.107,177.3551,-3.2201,-8762.2261
C00817=52.057,77.939,51.802,173.3985,-2.6286,-8763.7397
C00818=50.345,74.091,51.229,173.0280,-0.9152,-8764.1962
C00819=48.181,70.226,50.084,175.4707,-0.5069,-8764.4534
C00820=46.331,66.751,48.618,-179.9953,0.0033,-8764.7640
C00821=45.309,63.858,47.218,-170.4927,3.4787,-8765.3567
C00822=45.731,61.299,46.215,-161.9462,29.9155,-8766.7241
C00823=48.234,58.511,45.818,-176.2690,38.8474,-8769.5007
C00824=50.999,56.061,45.801,179.7668,39.2376,-8772.2930
C00825=53.591,53.591,45.812,-180.0000,39.2305,-8775.0000
C00826=56.061,50.999,45.801,-179.7668,39.2376,-8777.7070
C00827=58.511,48.233,45.818,176.2686,38.8474,-8780.4999
C00828=61.299,45.731,46.215,161.9462,29.9155,-8783.2759
C00829=63.858,45.309,47.218,170.4927,3.4787,-8784.6433
C00830=66.751,46.331,48.618,179.9953,0.0033,-8785.2360
C00831=70.226,48.181,50.084,-175.4707,-0.5069,-8785.5466
C00832=74.091,50.345,51.229,-173.0280,-0.9152,-8785.8038
C00833=77.939,52.057,51.802,-173.3985,-2.6286,-8786.2603
C00834=82.136,51.776,52.107,-177.3551,-3.2201,-8787.7739
C00835=86.092,49.437,52.356,-179.3324,-2.0949,-8790.1341
C00836=89.019,45.419,52.610,-179.9959,-0.1307,-8792.9686
C00837=91.330,40.710,52.777,179.9982,-0.0180,-8795.9753
C00838=93.367,35.794,52.777,179.9992,-0.0181,-8799.0247
C00839=95.062,30.830,52.610,179.9993,-0.1323,-8802.0314
C00840=95.834,25.919,52.356,179.3271,-2.0919,-8804.8660
C00841=94.690,21.467,52.107,177.3556,-3.2253,-8807.2265
C00842=91.921,18.302,51.802,173.3993,-2.6344,-8808.7393
C00843=87.989,16.791,51.229,173.0243,-0.9189,-8809.1961
C00844=83.726,15.588,50.084,175.4718,-0.5058,-8809.4535
C00845=79.961,14.439,48.618,-179.9944,-0.0010,-8809.7641
C00846=77.193,13.116,47.218,-170.4942,3.4778,-8810.3569
C00847=75.681,11.008,46.215,-161.9441,29.9170,-8811.7242
C00848=75.480,7.267,45.818,-176.2657,38.8470,-8814.5007
C00849=75.703,3.580,45.801,179.7689,39.2394,-8817.2925
C00850=75.789,0.000,45.812,-180.0000,39.2289,-8820.0000
C00851=75.703,-3.580,45.801,-179.7689,39.2394,-8822.7075
C00852=75.480,-7.267,45.818,176.2657,38.8470,-8825.4993
C00853=75.681,-11.008,46.215,161.9441,29.9170,-8828.2758
C00854=77.193,-13.116,47.218,170.4942,3.4778,-8829.6431
C00855=79.961,-14.439,48.618,179.9944,-0.0010,-8830.2359
C00856=83.726,-15.588,50.084,-175.4718,-0.5058,-8830.5465
C00857=87.989,-16.791,51.229,-173.0243,-0.9189,-8830.8039
C00858=91.921,-18.302,51.802,-173.3993,-2.6344,-8831.2607
C00859=94.690,-21.467,52.107,-177.3556,-3.2253,-8832.7735
C00860=95.834,-25.919,52.356,-179.3271,-2.0919,-8835.1340
C00861=95.062,-30.830,52.610,-179.9993,-0.1323,-8837.9686
C00862=93.367,-35.794,52.777,-179.9992,-0.0181,-8840.9753
C00863=91.330,-40.710,52.777,-179.9982,-0.0180,-8844.0247
C00864=89.019,-45.419,52.610,179.9959,-0.1307,-8847.0314
C00865=86.092,-49.437,52.356,179.3324,-2.0949,-8849.8659
C00866=82.136,-51.776,52.107,177.3551,-3.2201,-8852.2261
C00867=77.939,-52.057,51.802,173.3985,-2.6286,-8853.7397
C00868=74.091,-50.345,51.229,173.0280,-0.9152,-8854.1962
C00869=70.226,-48.181,50.084,175.4707,-0.5069,-8854.4534
C00870=66.751,-46.331,48.618,-179.9953,0.0033,-8854.7640
C00871=63.858,-45.309,47.218,-170.4927,3.4787,-8855.3567
C00872=61.299,-45.731,46.215,-161.9462,29.9155,-8856.7241
C00873=58.511,-48.234,45.818,-176.2690,38.8474,-8859.5007
C00874=56.061,-50.999,45.801,179.7668,39.2376,-8862.2930
C00875=53.591,-53.591,45.812,180.0000,39.2305,-8865.0000
C00876=50.999,-56.061,45.801,-179.7668,39.2376,-8867.7070
C00877=48.233,-58.511,45.818,176.2686,38.8474,-8870.4999
C00878=45.731,-61.299,46.215,161.9462,29.9155,-8873.2759
C00879=45.309,-63.858,47.218,170.4927,3.4787,-8874.6433
C00880=46.331,-66.751,48.618,179.9953,0.0033,-8875.2360
C00881=48.181,-70.226,50.084,-175.4707,-0.5069,-8875.5466
C00882=50.345,-74.091,51.229,-173.0280,-0.9152,-8875.8038
C00883=52.057,-77.939,51.802,-173.3985,-2.6286,-8876.2603
C00884=51.776,-82.136,52.107,-177.3551,-3.2201,-8877.7739
C00885=49.437,-86.092,52.356,-179.3324,-2.0949,-8880.1341
C00886=45.419,-89.019,52.610,-179.9959,-0.1307,-8882.9686
C00887=40.710,-91.330,52.777,179.9982,-0.0180,-8885.9753
C00888=35.794,-93.367,52.777,179.9992,-0.0181,-8889.0247
C00889=30.830,-95.062,52.610,179.9993,-0.1323,-8892.0314
C00890=25.919,-95.834,52.356,179.3271,-2.0919,-8894.8660
C00891=21.467,-94.690,52.107,177.3556,-3.2253,-8897.2265
C00892=18.302,-91.921,51.802,173.3993,-2.6344,-8898.7393
C00893=16.791,-87.989,51.229,173.0243,-0.9189,-8899.1961
C00894=15.588,-83.726,50.084,175.4718,-0.5058,-8899.4535
C00895=14.439,-79.961,48.618,-179.9944,-0.0010,-8899.7641
C00896=13.116,-77.193,47.218,-170.4942,3.4778,-8900.3569
C00897=11.008,-75.681,46.215,-161.9441,29.9170,-8901.7242
C00898=7.267,-75.480,45.818,-176.2657,38.8470,-8904.5007
C00899=3.580,-75.703,45.801,179.7689,39.2394,-8907.2925
C00900=0.000,-75.789,45.812,180.0000,39.2289,-8910.0000
C00901=-3.580,-75.703,45.801,-179.7689,39.2394,-8912.7075
C00902=-7.267,-75.480,45.818,176.2657,38.8470,-8915.4993
C00903=-11.008,-75.681,46.215,161.9441,29.9170,-8918.2758
C00904=-13.116,-77.193,47.218,170.4942,3.4778,-8919.6431
C00905=-14.439,-79.961,48.618,179.9944,-0.0010,-8920.2359
C00906=-15.588,-83.726,50.084,-175.4718,-0.5058,-8920.5465
C00907=-16.791,-87.989,51.229,-173.0243,-0.9189,-8920.8039
C00908=-18.302,-91.921,51.802,-173.3993,-2.6344,-8921.2607
C00909=-21.467,-94.690,52.107,-177.3556,-3.2253,-8922.7735
C00910=-25.919,-95.834,52.356,-179.3271,-2.0919,-8925.1340
C00911=-30.830,-95.062,52.610,-179.9993,-0.1323,-8927.9686
C00912=-35.794,-93.367,52.777,-179.9992,-0.0181,-8930.9753
C00913=-40.710,-91.330,52.777,-179.9982,-0.0180,-8934.0247
C00914=-45.419,-89.019,52.610,179.9959,-0.1307,-8937.0314
C00915=-49.437,-86.092,52.356,179.3324,-2.0949,-8939.8659
C00916=-51.776,-82.136,52.107,177.3551,-3.2201,-8942.2261
C00917=-52.057,-77.939,51.802,173.3985,-2.6286,-8943.7397
C00918=-50.345,-74.091,51.229,173.0280,-0.9152,-8944.1962
C00919=-48.181,-70.226,50.084,175.4707,-0.5069,-8944.4534
C00920=-46.331,-66.751,48.618,-179.9953,0.0033,-8944.7640
C00921=-45.309,-63.858,47.218,-170.4927,3.4787,-8945.3567
C00922=-45.731,-61.299,46.215,-161.9462,29.9155,-8946.7241
C00923=-48.234,-58.511,45.818,-176.2690,38.8474,-8949.5007
C00924=-50.999,-56.061,45.801,179.7668,39.2376,-8952.2930
C00925=-53.591,-53.591,45.812,180.0000,39.2305,-8955.0000
C00926=-56.061,-50.999,45.801,-179.7668,39.2376,-8957.7070
C00927=-58.511,-48.233,45.818,176.2686,38.8474,-8960.4999
C00928=-61.299,-45.731,46.215,161.9462,29.9155,-8963.2759
C00929=-63.858,-45.309,47.218,170.4927,3.4787,-8964.6433
C00930=-66.751,-46.331,48.618,179.9953,0.0033,-8965.2360
C00931=-70.226,-48.181,50.084,-175.4707,-0.5069,-8965.5466
C00932=-74.091,-50.345,51.229,-173.0280,-0.9152,-8965.8038
C00933=-77.939,-52.057,51.802,-173.3985,-2.6286,-8966.2603
C00934=-82.136,-51.776,52.107,-177.3551,-3.2201,-8967.7739
C00935=-86.092,-49.437,52.356,-179.3324,-2.0949,-8970.1341
C00936=-89.019,-45.419,52.610,-179.9959,-0.1307,-8972.9686
C00937=-91.330,-40.710,52.777,179.9982,-0.0180,-8975.9753
C00938=-93.367,-35.794,52.777,179.9992,-0.0181,-8979.0247
C00939=-95.062,-30.830,52.610,179.9993,-0.1323,-8982.0314
C00940=-95.834,-25.919,52.356,179.3271,-2.0919,-8984.8660
C00941=-94.690,-21.467,52.107,177.3556,-3.2253,-8987.2265
C00942=-91.921,-18.302,51.802,173.3993,-2.6344,-8988.7393
C00943=-87.989,-16.791,51.229,173.0243,-0.9189,-8989.1961
C00944=-83.726,-15.588,50.084,175.4718,-0.5058,-8989.4535
C00945=-79.961,-14.439,48.618,-179.9944,-0.0010,-8989.7641
C00946=-77.193,-13.116,47.218,-170.4942,3.4778,-8990.3569
C00947=-75.681,-11.008,46.215,-161.9441,29.9170,-8991.7242
C00948=-75.480,-7.267,45.818,-176.2657,38.8470,-8994.5007
C00949=-75.703,-3.580,45.801,179.7689,39.2394,-8997.2925
C00950=-75.789,0.000,45.812,180.0000,39.2289,-9000.0000
C00951=-75.703,3.580,45.801,-179.7689,39.2394,-9002.7075
C00952=-75.480,7.267,45.818,176.2657,38.8470,-9005.4993
C00953=-75.681,11.008,46.215,161.9441,29.9170,-9008.2758
C00954=-77.193,13.116,47.218,170.4942,3.4778,-9009.6431
C00955=-79.961,14.439,48.618,179.9944,-0.0010,-9010.2359
C00956=-83.726,15.588,50.084,-175.4718,-0.5058,-9010.5465
C00957=-87.989,16.791,51.229,-173.0243,-0.9189,-9010.8039
C00958=-91.921,18.302,51.802,-173.3993,-2.6344,-9011.2607
C00959=-94.690,21.467,52.107,-177.3556,-3.2253,-9012.7735
C00960=-95.834,25.919,52.356,-179.3271,-2.0919,-9015.1340
C00961=-95.062,30.830,52.610,-179.9993,-0.1323,-9017.9686
C00962=-93.367,35.794,52.777,-179.9992,-0.0181,-9020.9753
C00963=-91.330,40.710,52.777,-179.9982,-0.0180,-9024.0247
C00964=-89.019,45.419,52.610,179.9959,-0.1307,-9027.0314
C00965=-86.092,49.437,52.356,179.3324,-2.0949,-9029.8659
C00966=-82.136,51.776,52.107,177.3551,-3.2201,-9032.2261
C00967=-77.939,52.057,51.802,173.3985,-2.6286,-9033.7397
C00968=-74.091,50.345,51.229,173.0280,-0.9152,-9034.1962
C00969=-70.226,48.181,50.084,175.4707,-0.5069,-9034.4534
C00970=-66.751,46.331,48.618,-179.9953,0.0033,-9034.7640
C00971=-63.858,45.309,47.218,-170.4927,3.4787,-9035.3567
C00972=-61.299,45.731,46.215,-161.9462,29.9155,-9036.7241
C00973=-58.511,48.234,45.818,-176.2690,38.8474,-9039.5007
C00974=-56.061,50.999,45.801,179.7668,39.2376,-9042.2930
C00975=-53.591,53.591,45.812,-180.0000,39.2305,-9045.0000
C00976=-50.999,56.061,45.801,-179.7668,39.2376,-9047.7070
C00977=-48.233,58.511,45.818,176.2686,38.8474,-9050.4999
C00978=-45.731,61.299,46.215,161.9462,29.9155,-9053.2759
C00979=-45.309,63.858,47.218,170.4927,3.4787,-9054.6433
C00980=-46.331,66.751,48.618,179.9953,0.0033,-9055.2360
C00981=-48.181,70.226,50.084,-175.4707,-0.5069,-9055.5466
C00982=-50.345,74.091,51.229,-173.0280,-0.9152,-9055.8038
C00983=-52.057,77.939,51.802,-173.3985,-2.6286,-9056.2603
C00984=-51.776,82.136,52.107,-177.3551,-3.2201,-9057.7739
C00985=-49.437,86.092,52.356,-179.3324,-2.0949,-9060.1341
C00986=-45.419,89.019,52.610,-179.9959,-0.1307,-9062.9686
C00987=-40.710,91.330,52.777,179.9982,-0.0180,-9065.9753
C00988=-35.794,93.367,52.777,179.9992,-0.0181,-9069.0247
C00989=-30.830,95.062,52.610,179.9993,-0.1323,-9072.0314
C00990=-25.919,95.834,52.356,179.3271,-2.0919,-9074.8660
C00991=-21.467,94.690,52.107,177.3556,-3.2253,-9077.2265
C00992=-18.302,91.921,51.802,173.3993,-2.6344,-9078.7393
C00993=-16.791,87.989,51.229,173.0243,-0.9189,-9079.1961
C00994=-15.588,83.726,50.084,175.4718,-0.5058,-9079.4535
C00995=-14.439,79.961,48.618,-179.9944,-0.0010,-9079.7641
C00996=-13.116,77.193,47.218,-170.4942,3.4778,-9080.3569
C00997=-11.008,75.681,46.215,-161.9441,29.9170,-9081.7242
C00998=-7.267,75.480,45.818,-176.2657,38.8470,-9084.5007
C00999=-3.580,75.703,45.801,179.7689,39.2394,-9087.2925
C01000=0.000,74.396,47.516,-180.0000,39.2862,-9090.0000
C01001=3.453,74.315,47.503,-179.7551,39.2958,-9092.6603
C01002=7.053,74.105,47.522,175.9830,38.8590,-9095.4368
C01003=10.745,74.349,47.946,161.3656,28.9678,-9098.2235
C01004=12.792,75.972,49.019,171.7820,2.6538,-9099.5577
C01005=14.064,78.919,50.519,-179.2168,-0.1165,-9100.1045
C01006=15.177,82.922,52.090,-175.0027,-0.4746,-9100.3719
C01007=16.346,87.459,53.317,-172.6692,-0.8205,-9100.5864
C01008=17.816,91.657,53.931,-172.9897,-2.5671,-9100.9998
C01009=21.009,94.635,54.258,-177.1190,-3.3590,-9102.5167
C01010=25.555,95.900,54.525,-179.2765,-2.1798,-9104.9212
C01011=30.600,95.138,54.796,-179.9978,-0.1377,-9107.8298
C01012=35.715,93.397,54.976,-179.9992,-0.0181,-9110.9268
C01013=40.787,91.296,54.976,-179.9982,-0.0180,-9114.0730
C01014=45.636,88.910,54.796,179.9989,-0.1358,-9117.1707
C01015=49.741,85.881,54.525,179.2809,-2.1781,-9120.0788
C01016=52.061,81.773,54.258,177.1161,-3.3597,-9122.4830
C01017=52.213,77.409,53.931,172.9890,-2.5623,-9124.0000
C01018=50.285,73.401,53.317,172.6678,-0.8206,-9124.4140
C01019=47.903,69.367,52.090,175.0015,-0.4761,-9124.6279
C01020=45.859,65.749,50.519,179.2140,-0.1151,-9124.8952
C01021=44.675,62.766,49.019,-171.7766,2.6554,-9125.4421
C01022=44.975,60.171,47.946,-161.3601,28.9675,-9126.7764
C01023=47.412,57.387,47.522,-175.9840,38.8604,-9129.5628
C01024=50.108,54.990,47.503,179.7517,39.2962,-9132.3404
C01025=52.606,52.606,47.516,-180.0000,39.2837,-9135.0000
C01026=54.990,50.108,47.503,-179.7517,39.2962,-9137.6596
C01027=57.387,47.412,47.522,175.9840,38.8604,-9140.4372
C01028=60.171,44.975,47.946,161.3638,28.9717,-9143.2236
C01029=62.766,44.675,49.019,171.7766,2.6554,-9144.5579
C01030=65.749,45.859,50.519,-179.2140,-0.1151,-9145.1048
C01031=69.367,47.903,52.090,-175.0015,-0.4761,-9145.3721
C01032=73.401,50.285,53.317,-172.6678,-0.8206,-9145.5860
C01033=77.409,52.213,53.931,-172.9890,-2.5623,-9146.0000
C01034=81.773,52.061,54.258,-177.1161,-3.3597,-9147.5170
C01035=85.881,49.741,54.525,-179.2809,-2.1781,-9149.9212
C01036=88.910,45.636,54.796,-179.9989,-0.1358,-9152.8293
C01037=91.296,40.787,54.976,179.9982,-0.0180,-9155.9270
C01038=93.397,35.715,54.976,179.9992,-0.0181,-9159.0732
C01039=95.138,30.600,54.796,179.9978,-0.1377,-9162.1702
C01040=95.900,25.555,54.525,179.2765,-2.1798,-9165.0788
C01041=94.635,21.009,54.258,177.1190,-3.3590,-9167.4833
C01042=91.657,17.816,53.931,172.9897,-2.5671,-9169.0002
C01043=87.459,16.346,53.317,172.6692,-0.8205,-9169.4136
C01044=82.922,15.177,52.090,175.0027,-0.4746,-9169.6281
C01045=78.919,14.064,50.519,179.2168,-0.1165,-9169.8955
C01046=75.972,12.792,49.019,-171.7820,2.6538,-9170.4423
C01047=74.349,10.745,47.946,-161.3656,28.9678,-9171.7765
C01048=74.105,7.053,47.522,-175.9830,38.8590,-9174.5632
C01049=74.315,3.453,47.503,179.7551,39.2958,-9177.3397
C01050=74.396,0.000,47.516,-180.0000,39.2862,-9180.0000
C01051=74.315,-3.453,47.503,-179.7551,39.2958,-9182.6603
C01052=74.105,-7.053,47.522,175.9830,38.8590,-9185.4368
C01053=74.349,-10.745,47.946,161.3656,28.9678,-9188.2235
C01054=75.972,-12.792,49.019,171.7820,2.6538,-9189.5577
C01055=78.919,-14.064,50.519,-179.2168,-0.1165,-9190.1045
C01056=82.922,-15.177,52.090,-175.0027,-0.4746,-9190.3719
C01057=87.459,-16.346,53.317,-172.6692,-0.8205,-9190.5864
C01058=91.657,-17.816,53.931,-172.9897,-2.5671,-9190.9998
C01059=94.635,-21.009,54.258,-177.1190,-3.3590,-9192.5167
C01060=95.900,-25.555,54.525,-179.2765,-2.1798,-9194.9212
C01061=95.138,-30.600,54.796,-179.9978,-0.1377,-9197.8298
C01062=93.397,-35.715,54.976,-179.9992,-0.0181,-9200.9268
C01063=91.296,-40.787,54.976,-179.9982,-0.0180,-9204.0730
C01064=88.910,-45.636,54.796,179.9989,-0.1358,-9207.1707
C01065=85.881,-49.741,54.525,179.2809,-2.1781,-9210.0788
C01066=81.773,-52.061,54.258,177.1161,-3.3597,-9212.4830
C01067=77.409,-52.213,53.931,172.9890,-2.5623,-9214.0000
C01068=73.401,-50.285,53.317,172.6678,-0.8206,-9214.4140
C01069=69.367,-47.903,52.090,175.0015,-0.4761,-9214.6279
C01070=65.749,-45.859,50.519,179.2140,-0.1151,-9214.8952
C01071=62.766,-44.675,49.019,-171.7766,2.6554,-9215.4421
C01072=60.171,-44.975,47.946,-161.3601,28.9675,-9216.7764
C01073=57.387,-47.412,47.522,-175.9840,38.8604,-9219.5628
C01074=54.990,-50.108,47.503,179.7517,39.2962,-9222.3404
C01075=52.606,-52.606,47.516,-180.0000,39.2837,-9225.0000
C01076=50.108,-54.990,47.503,-179.7517,39.2962,-9227.6596
C01077=47.412,-57.387,47.522,175.9840,38.8604,-9230.4372
C01078=44.975,-60.171,47.946,161.3638,28.9717,-9233.2236
C01079=44.675,-62.766,49.019,171.7766,2.6554,-9234.5579
C01080=45.859,-65.749,50.519,-179.2140,-0.1151,-9235.1048
C01081=47.903,-69.367,52.090,-175.0015,-0.4761,-9235.3721
C01082=50.285,-73.401,53.317,-172.6678,-0.8206,-9235.5860
C01083=52.213,-77.409,53.931,-172.9890,-2.5623,-9236.0000
C01084=52.061,-81.773,54.258,-177.1161,-3.3597,-9237.5170
C01085=49.741,-85.881,54.525,-179.2809,-2.1781,-9239.9212
C01086=45.636,-88.910,54.796,-179.9989,-0.1358,-9242.8293
C01087=40.787,-91.296,54.976,179.9982,-0.0180,-9245.9270
C01088=35.715,-93.397,54.976,179.9992,-0.0181,-9249.0732
C01089=30.600,-95.138,54.796,179.9978,-0.1377,-9252.1702
C01090=25.555,-95.900,54.525,179.2765,-2.1798,-9255.0788
C01091=21.009,-94.635,54.258,177.1190,-3.3590,-9257.4833
C01092=17.816,-91.657,53.931,172.9897,-2.5671,-9259.0002
C01093=16.346,-87.459,53.317,172.6692,-0.8205,-9259.4136
C01094=15.177,-82.922,52.090,175.0027,-0.4746,-9259.6281
C01095=14.064,-78.919,50.519,179.2168,-0.1165,-9259.8955
C01096=12.792,-75.972,49.019,-171.7820,2.6538,-9260.4423
C01097=10.745,-74.349,47.946,-161.3656,28.9678,-9261.7765
C01098=7.053,-74.105,47.522,-175.9830,38.8590,-9264.5632
C01099=3.453,-74.315,47.503,179.7551,39.2958,-9267.3397
C01100=0.000,-74.396,47.516,-180.0000,39.2862,-9270.0000
C01101=-3.453,-74.315,47.503,-179.7551,39.2958,-9272.6603
C01102=-7.053,-74.105,47.522,175.9830,38.8590,-9275.4368
C01103=-10.745,-74.349,47.946,161.3656,28.9678,-9278.2235
C01104=-12.792,-75.972,49.019,171.7820,2.6538,-9279.5577
C01105=-14.064,-78.919,50.519,-179.2168,-0.1165,-9280.1045
C01106=-15.177,-82.922,52.090,-175.0027,-0.4746,-9280.3719
C01107=-16.346,-87.459,53.317,-172.6692,-0.8205,-9280.5864
C01108=-17.816,-91.657,53.931,-172.9897,-2.5671,-9280.9998
C01109=-21.009,-94.635,54.258,-177.1190,-3.3590,-9282.5167
C01110=-25.555,-95.900,54.525,-179.2765,-2.1798,-9284.9212
C01111=-30.600,-95.138,54.796,-179.9978,-0.1377,-9287.8298
C01112=-35.715,-93.397,54.976,-179.9992,-0.0181,-9290.9268
C01113=-40.787,-91.296,54.976,-179.9982,-0.0180,-9294.0730
C01114=-45.636,-88.910,54.796,179.9989,-0.1358,-9297.1707
C01115=-49.741,-85.881,54.525,179.2809,-2.1781,-9300.0788
C01116=-52.061,-81.773,54.258,177.1161,-3.3597,-9302.4830
C01117=-52.213,-77.409,53.931,172.9890,-2.5623,-9304.0000
C01118=-50.285,-73.401,53.317,172.6678,-0.8206,-9304.4140
C01119=-47.903,-69.367,52.090,175.0015,-0.4761,-9304.6279
C01120=-45.859,-65.749,50.519,179.2140,-0.1151,-9304.8952
C01121=-44.675,-62.766,49.019,-171.7766,2.6554,-9305.4421
C01122=-44.975,-60.171,47.946,-161.3601,28.9675,-9306.7764
C01123=-47.412,-57.387,47.522,-175.9840,38.8604,-9309.5628
C01124=-50.108,-54.990,47.503,179.7517,39.2962,-9312.3404
C01125=-52.606,-52.606,47.516,180.0000,39.2837,-9315.0000
C01126=-54.990,-50.108,47.503,-179.7517,39.2962,-9317.6596
C01127=-57.387,-47.412,47.522,175.9840,38.8604,-9320.4372
C01128=-60.171,-44.975,47.946,161.3638,28.9717,-9323.2236
C01129=-62.766,-44.675,49.019,171.7766,2.6554,-9324.5579
C01130=-65.749,-45.859,50.519,-179.2140,-0.1151,-9325.1048
C01131=-69.367,-47.903,52.090,-175.0015,-0.4761,-9325.3721
C01132=-73.401,-50.285,53.317,-172.6678,-0.8206,-9325.5860
C01133=-77.409,-52.213,53.931,-172.9890,-2.5623,-9326.0000
C01134=-81.773,-52.061,54.258,-177.1161,-3.3597,-9327.5170
C01135=-85.881,-49.741,54.525,-179.2809,-2.1781,-9329.9212
C01136=-88.910,-45.636,54.796,-179.9989,-0.1358,-9332.8293
C01137=-91.296,-40.787,54.976,179.9982,-0.0180,-9335.9270
C01138=-93.397,-35.715,54.976,179.9992,-0.0181,-9339.0732
C01139=-95.138,-30.600,54.796,179.9978,-0.1377,-9342.1702
C01140=-95.900,-25.555,54.525,179.2765,-2.1798,-9345.0788
C01141=-94.635,-21.009,54.258,177.1190,-3.3590,-9347.4833
C01142=-91.657,-17.816,53.931,172.9897,-2.5671,-9349.0002
C01143=-87.459,-16.346,53.317,172.6692,-0.8205,-9349.4136
C01144=-82.922,-15.177,52.090,175.0027,-0.4746,-9349.6281
C01145=-78.919,-14.064,50.519,179.2168,-0.1165,-9349.8955
C01146=-75.972,-12.792,49.019,-171.7820,2.6538,-9350.4423
C01147=-74.349,-10.745,47.946,-161.3656,28.9678,-9351.7765
C01148=-74.105,-7.053,47.522,-175.9830,38.8590,-9354.5632
C01149=-74.315,-3.453,47.503,179.7551,39.2958,-9357.3397
C01150=-74.396,0.000,47.516,180.0000,39.2862,-9360.0000
C01151=-74.315,3.453,47.503,-179.7551,39.2958,-9362.6603
C01152=-74.105,7.053,47.522,175.9830,38.8590,-9365.4368
C01153=-74.349,10.745,47.946,161.3656,28.9678,-9368.2235
C01154=-75.972,12.792,49.019,171.7820,2.6538,-9369.5577
C01155=-78.919,14.064,50.519,-179.2168,-0.1165,-9370.1045
C01156=-82.922,15.177,52.090,-175.0027,-0.4746,-9370.3719
C01157=-87.459,16.346,53.317,-172.6692,-0.8205,-9370.5864
C01158=-91.657,17.816,53.931,-172.9897,-2.5671,-9370.9998
C01159=-94.635,21.009,54.258,-177.1190,-3.3590,-9372.5167
C01160=-95.900,25.555,54.525,-179.2765,-2.1798,-9374.9212
C01161=-95.138,30.600,54.796,-179.9978,-0.1377,-9377.8298
C01162=-93.397,35.715,54.976,-179.9992,-0.0181,-9380.9268
C01163=-91.296,40.787,54.976,-179.9982,-0.0180,-9384.0730
C01164=-88.910,45.636,54.796,179.9989,-0.1358,-9387.1707
C01165=-85.881,49.741,54.525,179.2809,-2.1781,-9390.0788
C01166=-81.773,52.061,54.258,177.1161,-3.3597,-9392.4830
C01167=-77.409,52.213,53.931,172.9890,-2.5623,-9394.0000
C01168=-73.401,50.285,53.317,172.6678,-0.8206,-9394.4140
C01169=-69.367,47.903,52.090,175.0015,-0.4761,-9394.6279
C01170=-65.749,45.859,50.519,179.2140,-0.1151,-9394.8952
C01171=-62.766,44.675,49.019,-171.7766,2.6554,-9395.4421
C01172=-60.171,44.975,47.946,-161.3601,28.9675,-9396.7764
C01173=-57.387,47.412,47.522,-175.9840,38.8604,-9399.5628
C01174=-54.990,50.108,47.503,179.7517,39.2962,-9402.3404
C01175=-52.606,52.606,47.516,180.0000,39.2837,-9405.0000
C01176=-50.108,54.990,47.503,-179.7517,39.2962,-9407.6596
C01177=-47.412,57.387,47.522,175.9840,38.8604,-9410.4372
C01178=-44.975,60.171,47.946,161.3638,28.9717,-9413.2236
C01179=-44.675,62.766,49.019,171.7766,2.6554,-9414.5579
C01180=-45.859,65.749,50.519,-179.2140,-0.1151,-9415.1048
C01181=-47.903,69.367,52.090,-175.0015,-0.4761,-9415.3721
C01182=-50.285,73.401,53.317,-172.6678,-0.8206,-9415.5860
C01183=-52.213,77.409,53.931,-172.9890,-2.5623,-9416.0000
C01184=-52.061,81.773,54.258,-177.1161,-3.3597,-9417.5170
C01185=-49.741,85.881,54.525,-179.2809,-2.1781,-9419.9212
C01186=-45.636,88.910,54.796,-179.9989,-0.1358,-9422.8293
C01187=-40.787,91.296,54.976,179.9982,-0.0180,-9425.9270
C01188=-35.715,93.397,54.976,179.9992,-0.0181,-9429.0732
C01189=-30.600,95.138,54.796,179.9978,-0.1377,-9432.1702
C01190=-25.555,95.900,54.525,179.2765,-2.1798,-9435.0788
C01191=-21.009,94.635,54.258,177.1190,-3.3590,-9437.4833
C01192=-17.816,91.657,53.931,172.9897,-2.5671,-9439.0002
C01193=-16.346,87.459,53.317,172.6692,-0.8205,-9439.4136
C01194=-15.177,82.922,52.090,175.0027,-0.4746,-9439.6281
C01195=-14.064,78.919,50.519,179.2168,-0.1165,-9439.8955
C01196=-12.792,75.972,49.019,-171.7820,2.6538,-9440.4423
C01197=-10.745,74.349,47.946,-161.3656,28.9678,-9441.7765
C01198=-7.053,74.105,47.522,-175.9830,38.8590,-9444.5632
C01199=-3.453,74.315,47.503,179.7551,39.2958,-9447.3397
C01200=0.000,73.003,49.219,180.0000,39.2701,-9450.0000
C01201=3.325,72.927,49.205,-179.7359,39.2790,-9452.6105
C01202=6.839,72.729,49.225,175.6988,38.7974,-9455.3720
C01203=10.483,73.017,49.677,160.9132,27.9152,-9458.1701
C01204=12.469,74.753,50.822,173.0334,1.9875,-9459.4699
C01205=13.691,77.880,52.422,-178.5184,-0.1876,-9459.9705
C01206=14.768,82.123,54.099,-174.6161,-0.4381,-9460.1944
C01207=15.905,86.934,55.407,-172.3962,-0.7222,-9460.3679
C01208=17.335,91.395,56.062,-172.6676,-2.4726,-9460.7398
C01209=20.556,94.581,56.410,-176.9158,-3.4545,-9462.2618
C01210=25.196,95.965,56.695,-179.2377,-2.2474,-9464.7112
C01211=30.373,95.213,56.983,-179.9964,-0.1432,-9467.6927
C01212=35.638,93.426,57.174,-179.9992,-0.0181,-9470.8797
C01213=40.862,91.262,57.174,-179.9982,-0.0180,-9474.1202
C01214=45.849,88.802,56.983,179.9967,-0.1435,-9477.3076
C01215=50.042,85.674,56.695,179.2339,-2.2461,-9480.2891
C01216=52.343,81.414,56.410,176.9125,-3.4589,-9482.7379
C01217=52.368,76.884,56.062,172.6714,-2.4710,-9484.2600
C01218=50.225,72.718,55.407,172.3996,-0.7206,-9484.6321
C01219=47.627,68.512,54.099,174.6158,-0.4388,-9484.8056
C01220=45.389,64.750,52.422,178.5149,-0.1874,-9485.0300
C01221=44.041,61.675,50.822,-173.0367,1.9870,-9485.5299
C01222=44.219,59.044,49.677,-160.9107,27.9123,-9486.8301
C01223=46.591,56.263,49.225,-175.6975,38.7970,-9489.6279
C01224=49.216,53.919,49.205,179.7373,39.2787,-9492.3891
C01225=51.621,51.621,49.219,-180.0000,39.2701,-9495.0000
C01226=53.919,49.216,49.205,-179.7373,39.2787,-9497.6109
C01227=56.263,46.591,49.225,175.6975,38.7970,-9500.3721
C01228=59.044,44.219,49.677,160.9107,27.9123,-9503.1699
C01229=61.675,44.041,50.822,173.0367,1.9870,-9504.4701
C01230=64.750,45.389,52.422,-178.5149,-0.1874,-9504.9700
C01231=68.512,47.627,54.099,-174.6158,-0.4388,-9505.1944
C01232=72.718,50.225,55.407,-172.3996,-0.7206,-9505.3679
C01233=76.884,52.368,56.062,-172.6714,-2.4710,-9505.7400
C01234=81.414,52.343,56.410,-176.9125,-3.4589,-9507.2621
C01235=85.674,50.042,56.695,-179.2339,-2.2461,-9509.7109
C01236=88.802,45.849,56.983,-179.9967,-0.1435,-9512.6924
C01237=91.262,40.862,57.174,179.9982,-0.0180,-9515.8798
C01238=93.426,35.638,57.174,179.9992,-0.0181,-9519.1203
C01239=95.213,30.373,56.983,179.9964,-0.1432,-9522.3073
C01240=95.965,25.196,56.695,179.2377,-2.2474,-9525.2888
C01241=94.581,20.556,56.410,176.9158,-3.4545,-9527.7382
C01242=91.395,17.335,56.062,172.6676,-2.4726,-9529.2602
C01243=86.934,15.905,55.407,172.3962,-0.7222,-9529.6321
C01244=82.123,14.768,54.099,174.6161,-0.4381,-9529.8056
C01245=77.880,13.691,52.422,178.5184,-0.1876,-9530.0295
C01246=74.753,12.469,50.822,-173.0334,1.9875,-9530.5301
C01247=73.017,10.483,49.677,-160.9132,27.9152,-9531.8299
C01248=72.729,6.839,49.225,-175.6988,38.7974,-9534.6280
C01249=72.927,3.325,49.205,179.7359,39.2790,-9537.3895
C01250=73.003,0.000,49.219,-180.0000,39.2701,-9540.0000
C01251=72.927,-3.325,49.205,-179.7359,39.2790,-9542.6105
C01252=72.729,-6.839,49.225,175.6988,38.7974,-9545.3720
C01253=73.017,-10.483,49.677,160.9132,27.9152,-9548.1701
C01254=74.753,-12.469,50.822,173.0334,1.9875,-9549.4699
C01255=77.880,-13.691,52.422,-178.5184,-0.1876,-9549.9705
C01256=82.123,-14.768,54.099,-174.6161,-0.4381,-9550.1944
C01257=86.934,-15.905,55.407,-172.3962,-0.7222,-9550.3679
C01258=91.395,-17.335,56.062,-172.6676,-2.4726,-9550.7398
C01259=94.581,-20.556,56.410,-176.9158,-3.4545,-9552.2618
C01260=95.965,-25.196,56.695,-179.2377,-2.2474,-9554.7112
C01261=95.213,-30.373,56.983,-179.9964,-0.1432,-9557.6927
C01262=93.426,-35.638,57.174,-179.9992,-0.0181,-9560.8797
C01263=91.262,-40.862,57.174,-179.9982,-0.0180,-9564.1202
C01264=88.802,-45.849,56.983,179.9967,-0.1435,-9567.3076
C01265=85.674,-50.042,56.695,179.2339,-2.2461,-9570.2891
C01266=81.414,-52.343,56.410,176.9125,-3.4589,-9572.7379
C01267=76.884,-52.368,56.062,172.6714,-2.4710,-9574.2600
C01268=72.718,-50.225,55.407,172.3996,-0.7206,-9574.6321
C01269=68.512,-47.627,54.099,174.6158,-0.4388,-9574.8056
C01270=64.750,-45.389,52.422,178.5149,-0.1874,-9575.0300
C01271=61.675,-44.041,50.822,-173.0367,1.9870,-9575.5299
C01272=59.044,-44.219,49.677,-160.9107,27.9123,-9576.8301
C01273=56.263,-46.591,49.225,-175.6975,38.7970,-9579.6279
C01274=53.919,-49.216,49.205,179.7373,39.2787,-9582.3891
C01275=51.621,-51.621,49.219,-180.0000,39.2701,-9585.0000
C01276=49.216,-53.919,49.205,-179.7373,39.2787,-9587.6109
C01277=46.591,-56.263,49.225,175.6975,38.7970,-9590.3721
C01278=44.219,-59.044,49.677,160.9107,27.9123,-9593.1699
C01279=44.041,-61.675,50.822,173.0367,1.9870,-9594.4701
C01280=45.389,-64.750,52.422,-178.5149,-0.1874,-9594.9700
C01281=47.627,-68.512,54.099,-174.6158,-0.4388,-9595.1944
C01282=50.225,-72.718,55.407,-172.3996,-0.7206,-9595.3679
C01283=52.368,-76.884,56.062,-172.6714,-2.4710,-9595.7400
C01284=52.343,-81.414,56.410,-176.9125,-3.4589,-9597.2621
C01285=50.042,-85.674,56.695,-179.2339,-2.2461,-9599.7109
C01286=45.849,-88.802,56.983,-179.9967,-0.1435,-9602.6924
C01287=40.862,-91.262,57.174,179.9982,-0.0180,-9605.8798
C01288=35.638,-93.426,57.174,179.9992,-0.0181,-9609.1203
C01289=30.373,-95.213,56.983,179.9964,-0.1432,-9612.3073
C01290=25.196,-95.965,56.695,179.2377,-2.2474,-9615.2888
C01291=20.556,-94.581,56.410,176.9158,-3.4545,-9617.7382
C01292=17.335,-91.395,56.062,172.6676,-2.4726,-9619.2602
C01293=15.905,-86.934,55.407,172.3962,-0.7222,-9619.6321
C01294=14.768,-82.123,54.099,174.6161,-0.4381,-9619.8056
C01295=13.691,-77.880,52.422,178.5184,-0.1876,-9620.0295
C01296=12.469,-74.753,50.822,-173.0334,1.9875,-9620.5301
C01297=10.483,-73.017,49.677,-160.9132,27.9152,-9621.8299
C01298=6.839,-72.729,49.225,-175.6988,38.7974,-9624.6280
C01299=3.325,-72.927,49.205,179.7359,39.2790,-9627.3895
C01300=0.000,-73.003,49.219,-180.0000,39.2701,-9630.0000
C01301=-3.325,-72.927,49.205,-179.7359,39.2790,-9632.6105
C01302=-6.839,-72.729,49.225,175.6988,38.7974,-9635.3720
C01303=-10.483,-73.017,49.677,160.9132,27.9152,-9638.1701
C01304=-12.469,-74.753,50.822,173.0334,1.9875,-9639.4699
C01305=-13.691,-77.880,52.422,-178.5184,-0.1876,-9639.9705
C01306=-14.768,-82.123,54.099,-174.6161,-0.4381,-9640.1944
C01307=-15.905,-86.934,55.407,-172.3962,-0.7222,-9640.3679
C01308=-17.335,-91.395,56.062,-172.6676,-2.4726,-9640.7398
C01309=-20.556,-94.581,56.410,-176.9158,-3.4545,-9642.2618
C01310=-25.196,-95.965,56.695,-179.2377,-2.2474,-9644.7112
C01311=-30.373,-95.213,56.983,-179.9964,-0.1432,-9647.6927
C01312=-35.638,-93.426,57.174,-179.9992,-0.0181,-9650.8797
C01313=-40.862,-91.262,57.174,-179.9982,-0.0180,-9654.1202
C01314=-45.849,-88.802,56.983,179.9967,-0.1435,-9657.3076
C01315=-50.042,-85.674,56.695,179.2339,-2.2461,-9660.2891
C01316=-52.343,-81.414,56.410,176.9125,-3.4589,-9662.7379
C01317=-52.368,-76.884,56.062,172.6714,-2.4710,-9664.2600
C01318=-50.225,-72.718,55.407,172.3996,-0.7206,-9664.6321
C01319=-47.627,-68.512,54.099,174.6158,-0.4388,-9664.8056
C01320=-45.389,-64.750,52.422,178.5149,-0.1874,-9665.0300
C01321=-44.041,-61.675,50.822,-173.0367,1.9870,-9665.5299
C01322=-44.219,-59.044,49.677,-160.9107,27.9123,-9666.8301
C01323=-46.591,-56.263,49.225,-175.6975,38.7970,-9669.6279
C01324=-49.216,-53.919,49.205,179.7373,39.2787,-9672.3891
C01325=-51.621,-51.621,49.219,-180.0000,39.2701,-9675.0000
C01326=-53.919,-49.216,49.205,-179.7373,39.2787,-9677.6109
C01327=-56.263,-46.591,49.225,175.6975,38.7970,-9680.3721
C01328=-59.044,-44.219,49.677,160.9107,27.9123,-9683.1699
C01329=-61.675,-44.041,50.822,173.0367,1.9870,-9684.4701
C01330=-64.750,-45.389,52.422,-178.5149,-0.1874,-9684.9700
C01331=-68.512,-47.627,54.099,-174.6158,-0.4388,-9685.1944
C01332=-72.718,-50.225,55.407,-172.3996,-0.7206,-9685.3679
C01333=-76.884,-52.368,56.062,-172.6714,-2.4710,-9685.7400
C01334=-81.414,-52.343,56.410,-176.9125,-3.4589,-9687.2621
C01335=-85.674,-50.042,56.695,-179.2339,-2.2461,-9689.7109
C01336=-88.802,-45.849,56.983,-179.9967,-0.1435,-9692.6924
C01337=-91.262,-40.862,57.174,179.9982,-0.0180,-9695.8798
C01338=-93.426,-35.638,57.174,179.9992,-0.0181,-9699.1203
C01339=-95.213,-30.373,56.983,179.9964,-0.1432,-9702.3073
C01340=-95.965,-25.196,56.695,179.2377,-2.2474,-9705.2888
C01341=-94.581,-20.556,56.410,176.9158,-3.4545,-9707.7382
C01342=-91.395,-17.335,56.062,172.6676,-2.4726,-9709.2602
C01343=-86.934,-15.905,55.407,172.3962,-0.7222,-9709.6321
C01344=-82.123,-14.768,54.099,174.6161,-0.4381,-9709.8056
C01345=-77.880,-13.691,52.422,178.5184,-0.1876,-9710.0295
C01346=-74.753,-12.469,50.822,-173.0334,1.9875,-9710.5301
C01347=-73.017,-10.483,49.677,-160.9132,27.9152,-9711.8299
C01348=-72.729,-6.839,49.225,-175.6988,38.7974,-9714.6280
C01349=-72.927,-3.325,49.205,179.7359,39.2790,-9717.3895
C01350=-73.003,0.000,49.219,-180.0000,39.2701,-9720.0000
C01351=-72.927,3.325,49.205,-179.7359,39.2790,-9722.6105
C01352=-72.729,6.839,49.225,175.6988,38.7974,-9725.3720
C01353=-73.017,10.483,49.677,160.9132,27.9152,-9728.1701
C01354=-74.753,12.469,50.822,173.0334,1.9875,-9729.4699
C01355=-77.880,13.691,52.422,-178.5184,-0.1876,-9729.9705
C01356=-82.123,14.768,54.099,-174.6161,-0.4381,-9730.1944
C01357=-86.934,15.905,55.407,-172.3962,-0.7222,-9730.3679
C01358=-91.395,17.335,56.062,-172.6676,-2.4726,-9730.7398
C01359=-94.581,20.556,56.410,-176.9158,-3.4545,-9732.2618
C01360=-95.965,25.196,56.695,-179.2377,-2.2474,-9734.7112
C01361=-95.213,30.373,56.983,-179.9964,-0.1432,-9737.6927
C01362=-93.426,35.638,57.174,-179.9992,-0.0181,-9740.8797
C01363=-91.262,40.862,57.174,-179.9982,-0.0180,-9744.1202
C01364=-88.802,45.849,56.983,179.9967,-0.1435,-9747.3076
C01365=-85.674,50.042,56.695,179.2339,-2.2461,-9750.2891
C01366=-81.414,52.343,56.410,176.9125,-3.4589,-9752.7379
C01367=-76.884,52.368,56.062,172.6714,-2.4710,-9754.2600
C01368=-72.718,50.225,55.407,172.3996,-0.7206,-9754.6321
C01369=-68.512,47.627,54.099,174.6158,-0.4388,-9754.8056
C01370=-64.750,45.389,52.422,178.5149,-0.1874,-9755.0300
C01371=-61.675,44.041,50.822,-173.0367,1.9870,-9755.5299
C01372=-59.044,44.219,49.677,-160.9107,27.9123,-9756.8301
C01373=-56.263,46.591,49.225,-175.6975,38.7970,-9759.6279
C01374=-53.919,49.216,49.205,179.7373,39.2787,-9762.3891
C01375=-51.621,51.621,49.219,-180.0000,39.2701,-9765.0000
C01376=-49.216,53.919,49.205,-179.7373,39.2787,-9767.6109
C01377=-46.591,56.263,49.225,175.6975,38.7970,-9770.3721
C01378=-44.219,59.044,49.677,160.9107,27.9123,-9773.1699
C01379=-44.041,61.675,50.822,173.0367,1.9870,-9774.4701
C01380=-45.389,64.750,52.422,-178.5149,-0.1874,-9774.9700
C01381=-47.627,68.512,54.099,-174.6158,-0.4388,-9775.1944
C01382=-50.225,72.718,55.407,-172.3996,-0.7206,-9775.3679
C01383=-52.368,76.884,56.062,-172.6714,-2.4710,-9775.7400
C01384=-52.343,81.414,56.410,-176.9125,-3.4589,-9777.2621
C01385=-50.042,85.674,56.695,-179.2339,-2.2461,-9779.7109
C01386=-45.849,88.802,56.983,-179.9967,-0.1435,-9782.6924
C01387=-40.862,91.262,57.174,179.9982,-0.0180,-9785.8798
C01388=-35.638,93.426,57.174,179.9992,-0.0181,-9789.1203
C01389=-30.373,95.213,56.983,179.9964,-0.1432,-9792.3073
C01390=-25.196,95.965,56.695,179.2377,-2.2474,-9795.2888
C01391=-20.556,94.581,56.410,176.9158,-3.4545,-9797.7382
C01392=-17.335,91.395,56.062,172.6676,-2.4726,-9799.2602
C01393=-15.905,86.934,55.407,172.3962,-0.7222,-9799.6321
C01394=-14.768,82.123,54.099,174.6161,-0.4381,-9799.8056
C01395=-13.691,77.880,52.422,178.5184,-0.1876,-9800.0295
C01396=-12.469,74.753,50.822,-173.0334,1.9875,-9800.5301
C01397=-10.483,73.017,49.677,-160.9132,27.9152,-9801.8299
C01398=-6.839,72.729,49.225,-175.6988,38.7974,-9804.6280
C01399=-3.325,72.927,49.205,179.7359,39.2790,-9807.3895
C01400=0.000,71.612,50.923,180.0000,39.1761,-9810.0000
C01401=3.198,71.541,50.909,-179.7276,39.1884,-9812.5595
C01402=6.625,71.354,50.929,175.4226,38.6545,-9815.3045
C01403=10.220,71.688,51.410,160.5942,26.7641,-9818.1135
C01404=12.146,73.537,52.627,174.2333,1.4495,-9819.3788
C01405=13.319,76.847,54.328,-177.9012,-0.2296,-9819.8327
C01406=14.363,81.331,56.111,-174.3007,-0.3936,-9820.0151
C01407=15.469,86.415,57.500,-172.2051,-0.6229,-9820.1489
C01408=16.861,91.137,58.195,-172.4360,-2.3619,-9820.4816
C01409=20.110,94.527,58.564,-176.7443,-3.5170,-9822.0102
C01410=24.842,96.029,58.865,-179.1982,-2.2970,-9824.5040
C01411=30.149,95.287,59.171,179.9995,-0.1504,-9827.5575
C01412=35.562,93.456,59.373,-179.9992,-0.0181,-9830.8329
C01413=40.937,91.230,59.373,-179.9982,-0.0180,-9834.1669
C01414=46.059,88.697,59.171,179.9997,-0.1486,-9837.4422
C01415=50.337,85.469,58.865,179.2014,-2.2927,-9840.4960
C01416=52.621,81.060,58.564,176.7438,-3.5169,-9842.9901
C01417=52.521,76.366,58.195,172.4393,-2.3645,-9844.5184
C01418=50.167,72.043,57.500,172.2094,-0.6241,-9844.8513
C01419=47.354,67.666,56.111,174.3022,-0.3880,-9844.9851
C01420=44.921,63.757,54.328,177.8992,-0.2324,-9845.1672
C01421=43.410,60.587,52.627,-174.2351,1.4513,-9845.6212
C01422=43.464,57.918,51.410,-160.5947,26.7646,-9846.8860
C01423=45.770,55.140,50.929,-175.4250,38.6576,-9849.6950
C01424=48.325,52.849,50.909,179.7289,39.1881,-9852.4397
C01425=50.637,50.637,50.923,180.0000,39.1774,-9855.0000
C01426=52.848,48.326,50.909,-179.7280,39.1881,-9857.5591
C01427=55.140,45.770,50.930,175.4204,38.6542,-9860.3050
C01428=57.918,43.464,51.410,160.5947,26.7646,-9863.1140
C01429=60.587,43.410,52.627,174.2351,1.4513,-9864.3788
C01430=63.757,44.921,54.328,-177.8992,-0.2324,-9864.8328
C01431=67.666,47.354,56.111,-174.3022,-0.3880,-9865.0149
C01432=72.043,50.167,57.500,-172.2094,-0.6241,-9865.1487
C01433=76.366,52.521,58.195,-172.4393,-2.3645,-9865.4816
C01434=81.060,52.621,58.564,-176.7438,-3.5169,-9867.0099
C01435=85.469,50.337,58.865,-179.2014,-2.2927,-9869.5040
C01436=88.697,46.059,59.171,-179.9997,-0.1486,-9872.5578
C01437=91.230,40.937,59.373,179.9982,-0.0180,-9875.8331
C01438=93.456,35.562,59.373,179.9992,-0.0181,-9879.1671
C01439=95.287,30.149,59.171,-179.9995,-0.1504,-9882.4425
C01440=96.029,24.842,58.865,179.1982,-2.2970,-9885.4960
C01441=94.527,20.110,58.564,176.7443,-3.5170,-9887.9898
C01442=91.137,16.861,58.195,172.4360,-2.3619,-9889.5184
C01443=86.415,15.469,57.500,172.2051,-0.6229,-9889.8511
C01444=81.331,14.363,56.111,174.3007,-0.3936,-9889.9849
C01445=76.847,13.319,54.328,177.9012,-0.2296,-9890.1673
C01446=73.537,12.146,52.627,-174.2333,1.4495,-9890.6212
C01447=71.688,10.220,51.410,-160.5942,26.7641,-9891.8865
C01448=71.354,6.625,50.929,-175.4226,38.6545,-9894.6955
C01449=71.541,3.198,50.909,179.7276,39.1884,-9897.4405
C01450=71.612,0.000,50.923,180.0000,39.1761,-9900.0000
C01451=71.541,-3.198,50.909,-179.7276,39.1884,-9902.5595
C01452=71.354,-6.626,50.930,175.4219,38.6544,-9905.3053
C01453=71.688,-10.221,51.410,160.5938,26.7639,-9908.1143
C01454=73.537,-12.146,52.627,174.2333,1.4495,-9909.3788
C01455=76.847,-13.319,54.328,-177.9012,-0.2296,-9909.8327
C01456=81.331,-14.363,56.111,-174.3007,-0.3936,-9910.0151
C01457=86.415,-15.469,57.500,-172.2051,-0.6229,-9910.1489
C01458=91.137,-16.861,58.195,-172.4360,-2.3619,-9910.4816
C01459=94.527,-20.110,58.564,-176.7443,-3.5170,-9912.0102
C01460=96.029,-24.842,58.865,-179.1982,-2.2970,-9914.5040
C01461=95.287,-30.149,59.171,179.9995,-0.1504,-9917.5575
C01462=93.456,-35.562,59.373,-179.9992,-0.0181,-9920.8329
C01463=91.230,-40.937,59.373,-179.9982,-0.0180,-9924.1669
C01464=88.697,-46.059,59.171,179.9997,-0.1486,-9927.4422
C01465=85.469,-50.337,58.865,179.2014,-2.2927,-9930.4960
C01466=81.060,-52.621,58.564,176.7438,-3.5169,-9932.9901
C01467=76.366,-52.521,58.195,172.4393,-2.3645,-9934.5184
C01468=72.043,-50.167,57.500,172.2094,-0.6241,-9934.8513
C01469=67.666,-47.354,56.111,174.3022,-0.3880,-9934.9851
C01470=63.757,-44.921,54.328,177.8992,-0.2324,-9935.1672
C01471=60.587,-43.410,52.627,-174.2351,1.4513,-9935.6212
C01472=57.918,-43.464,51.410,-160.5947,26.7646,-9936.8860
C01473=55.140,-45.770,50.929,-175.4250,38.6576,-9939.6950
C01474=52.849,-48.325,50.909,179.7289,39.1881,-9942.4397
C01475=50.637,-50.637,50.923,180.0000,39.1774,-9945.0000
C01476=48.326,-52.848,50.909,-179.7280,39.1881,-9947.5591
C01477=45.770,-55.140,50.930,175.4204,38.6542,-9950.3050
C01478=43.464,-57.918,51.410,160.5947,26.7646,-9953.1140
C01479=43.410,-60.587,52.627,174.2351,1.4513,-9954.3788
C01480=44.921,-63.757,54.328,-177.8992,-0.2324,-9954.8328
C01481=47.354,-67.666,56.111,-174.3022,-0.3880,-9955.0149
C01482=50.167,-72.043,57.500,-172.2094,-0.6241,-9955.1487
C01483=52.521,-76.366,58.195,-172.4393,-2.3645,-9955.4816
C01484=52.621,-81.060,58.564,-176.7438,-3.5169,-9957.0099
C01485=50.337,-85.469,58.865,-179.2014,-2.2927,-9959.5040
C01486=46.059,-88.697,59.171,-179.9997,-0.1486,-9962.5578
C01487=40.937,-91.230,59.373,179.9982,-0.0180,-9965.8331
C01488=35.562,-93.456,59.373,179.9992,-0.0181,-9969.1671
C01489=30.149,-95.287,59.171,-179.9995,-0.1504,-9972.4425
C01490=24.842,-96.029,58.865,179.1982,-2.2970,-9975.4960
C01491=20.110,-94.527,58.564,176.7443,-3.5170,-9977.9898
C01492=16.861,-91.137,58.195,172.4360,-2.3619,-9979.5184
C01493=15.469,-86.415,57.500,172.2051,-0.6229,-9979.8511
C01494=14.363,-81.331,56.111,174.3007,-0.3936,-9979.9849
C01495=13.319,-76.847,54.328,177.9012,-0.2296,-9980.1673
C01496=12.146,-73.537,52.627,-174.2333,1.4495,-9980.6212
C01497=10.220,-71.688,51.410,-160.5942,26.7641,-9981.8865
C01498=6.625,-71.354,50.929,-175.4226,38.6545,-9984.6955
C01499=3.198,-71.541,50.909,179.7276,39.1884,-9987.4405
C01500=0.000,-71.612,50.923,-180.0000,39.1761,-9990.0000
C01501=-3.198,-71.541,50.909,-179.7276,39.1884,-9992.5595
C01502=-6.626,-71.354,50.930,175.4219,38.6544,-9995.3053
C01503=-10.221,-71.688,51.410,160.5938,26.7639,-9998.1143
C01504=-12.146,-73.537,52.627,174.2333,1.4495,-9999.3788
C01505=-13.319,-76.847,54.328,-177.9012,-0.2296,-9999.8327
C01506=-14.363,-81.331,56.111,-174.3007,-0.3936,-10000.0151
C01507=-15.469,-86.415,57.500,-172.2051,-0.6229,-10000.1489
C01508=-16.861,-91.137,58.195,-172.4360,-2.3619,-10000.4816
C01509=-20.110,-94.527,58.564,-176.7443,-3.5170,-10002.0102
C01510=-24.842,-96.029,58.865,-179.1982,-2.2970,-10004.5040
C01511=-30.149,-95.287,59.171,179.9995,-0.1504,-10007.5575
C01512=-35.562,-93.456,59.373,-179.9992,-0.0181,-10010.8329
C01513=-40.937,-91.230,59.373,-179.9982,-0.0180,-10014.1669
C01514=-46.059,-88.697,59.171,179.9997,-0.1486,-10017.4422
C01515=-50.337,-85.469,58.865,179.2014,-2.2927,-10020.4960
C01516=-52.621,-81.060,58.564,176.7438,-3.5169,-10022.9901
C01517=-52.521,-76.366,58.195,172.4393,-2.3645,-10024.5184
C01518=-50.167,-72.043,57.500,172.2094,-0.6241,-10024.8513
C01519=-47.354,-67.666,56.111,174.3022,-0.3880,-10024.9851
C01520=-44.921,-63.757,54.328,177.8992,-0.2324,-10025.1672
C01521=-43.410,-60.587,52.627,-174.2351,1.4513,-10025.6212
C01522=-43.464,-57.918,51.410,-160.5947,26.7646,-10026.8860
C01523=-45.770,-55.140,50.929,-175.4250,38.6576,-10029.6950
C01524=-48.325,-52.849,50.909,179.7289,39.1881,-10032.4397
C01525=-50.637,-50.637,50.923,-180.0000,39.1774,-10035.0000
C01526=-52.848,-48.326,50.909,-179.7280,39.1881,-10037.5591
C01527=-55.140,-45.770,50.930,175.4204,38.6542,-10040.3050
C01528=-57.918,-43.464,51.410,160.5947,26.7646,-10043.1140
C01529=-60.587,-43.410,52.627,174.2351,1.4513,-10044.3788
C01530=-63.757,-44.921,54.328,-177.8992,-0.2324,-10044.8328
C01531=-67.666,-47.354,56.111,-174.3022,-0.3880,-10045.0149
C01532=-72.043,-50.167,57.500,-172.2094,-0.6241,-10045.1487
C01533=-76.366,-52.521,58.195,-172.4393,-2.3645,-10045.4816
C01534=-81.060,-52.621,58.564,-176.7438,-3.5169,-10047.0099
C01535=-85.469,-50.337,58.865,-179.2014,-2.2927,-10049.5040
C01536=-88.697,-46.059,59.171,-179.9997,-0.1486,-10052.5578
C01537=-91.230,-40.937,59.373,179.9982,-0.0180,-10055.8331
C01538=-93.456,-35.562,59.373,179.9992,-0.0181,-10059.1671
C01539=-95.287,-30.149,59.171,-179.9995,-0.1504,-10062.4425
C01540=-96.029,-24.842,58.865,179.1982,-2.2970,-10065.4960
C01541=-94.527,-20.110,58.564,176.7443,-3.5170,-10067.9898
C01542=-91.137,-16.861,58.195,172.4360,-2.3619,-10069.5184
C01543=-86.415,-15.469,57.500,172.2051,-0.6229,-10069.8511
C01544=-81.331,-14.363,56.111,174.3007,-0.3936,-10069.9849
C01545=-76.847,-13.319,54.328,177.9012,-0.2296,-10070.1673
C01546=-73.537,-12.146,52.627,-174.2333,1.4495,-10070.6212
C01547=-71.688,-10.220,51.410,-160.5942,26.7641,-10071.8865
C01548=-71.354,-6.625,50.929,-175.4226,38.6545,-10074.6955
C01549=-71.541,-3.198,50.909,179.7276,39.1884,-10077.4405
C01550=-71.612,0.000,50.923,-180.0000,39.1761,-10080.0000
C01551=-71.541,3.198,50.909,-179.7276,39.1884,-10082.5595
C01552=-71.354,6.626,50.930,175.4219,38.6544,-10085.3053
C01553=-71.688,10.221,51.410,160.5938,26.7639,-10088.1143
C01554=-73.537,12.146,52.627,174.2333,1.4495,-10089.3788
C01555=-76.847,13.319,54.328,-177.9012,-0.2296,-10089.8327
C01556=-81.331,14.363,56.111,-174.3007,-0.3936,-10090.0151
C01557=-86.415,15.469,57.500,-172.2051,-0.6229,-10090.1489
C01558=-91.137,16.861,58.195,-172.4360,-2.3619,-10090.4816
C01559=-94.527,20.110,58.564,-176.7443,-3.5170,-10092.0102
C01560=-96.029,24.842,58.865,-179.1982,-2.2970,-10094.5040
C01561=-95.287,30.149,59.171,179.9995,-0.1504,-10097.5575
C01562=-93.456,35.562,59.373,-179.9992,-0.0181,-10100.8329
C01563=-91.230,40.937,59.373,-179.9982,-0.0180,-10104.1669
C01564=-88.697,46.059,59.171,179.9997,-0.1486,-10107.4422
C01565=-85.469,50.337,58.865,179.2014,-2.2927,-10110.4960
C01566=-81.060,52.621,58.564,176.7438,-3.5169,-10112.9901
C01567=-76.366,52.521,58.195,172.4393,-2.3645,-10114.5184
C01568=-72.043,50.167,57.500,172.2094,-0.6241,-10114.8513
C01569=-67.666,47.354,56.111,174.3022,-0.3880,-10114.9851
C01570=-63.757,44.921,54.328,177.8992,-0.2324,-10115.1672
C01571=-60.587,43.410,52.627,-174.2351,1.4513,-10115.6212
C01572=-57.918,43.464,51.410,-160.5947,26.7646,-10116.8860
C01573=-55.140,45.770,50.929,-175.4250,38.6576,-10119.6950
C01574=-52.849,48.325,50.909,179.7289,39.1881,-10122.4397
C01575=-50.637,50.637,50.923,-180.0000,39.1774,-10125.0000
C01576=-48.326,52.848,50.909,-179.7280,39.1881,-10127.5591
C01577=-45.770,55.140,50.930,175.4204,38.6542,-10130.3050
C01578=-43.464,57.918,51.410,160.5947,26.7646,-10133.1140
C01579=-43.410,60.587,52.627,174.2351,1.4513,-10134.3788
C01580=-44.921,63.757,54.328,-177.8992,-0.2324,-10134.8328
C01581=-47.354,67.666,56.111,-174.3022,-0.3880,-10135.0149
C01582=-50.167,72.043,57.500,-172.2094,-0.6241,-10135.1487
C01583=-52.521,76.366,58.195,-172.4393,-2.3645,-10135.4816
C01584=-52.621,81.060,58.564,-176.7438,-3.5169,-10137.0099
C01585=-50.337,85.469,58.865,-179.2014,-2.2927,-10139.5040
C01586=-46.059,88.697,59.171,-179.9997,-0.1486,-10142.5578
C01587=-40.937,91.230,59.373,179.9982,-0.0180,-10145.8331
C01588=-35.562,93.456,59.373,179.9992,-0.0181,-10149.1671
C01589=-30.149,95.287,59.171,-179.9995,-0.1504,-10152.4425
C01590=-24.842,96.029,58.865,179.1982,-2.2970,-10155.4960
C01591=-20.110,94.527,58.564,176.7443,-3.5170,-10157.9898
C01592=-16.861,91.137,58.195,172.4360,-2.3619,-10159.5184
C01593=-15.469,86.415,57.500,172.2051,-0.6229,-10159.8511
C01594=-14.363,81.331,56.111,174.3007,-0.3936,-10159.9849
C01595=-13.319,76.847,54.328,177.9012,-0.2296,-10160.1673
C01596=-12.146,73.537,52.627,-174.2333,1.4495,-10160.6212
C01597=-10.221,71.688,51.410,-160.5938,26.7639,-10161.8857
C01598=-6.626,71.354,50.930,-175.4219,38.6544,-10164.6947
C01599=-3.198,71.541,50.909,179.7276,39.1884,-10167.4405
C01600=0.000,70.224,52.630,-180.0000,39.0133,-10170.0000
C01601=3.072,70.158,52.615,-179.7154,39.0245,-10172.5072
C01602=6.412,69.984,52.637,175.1539,38.4339,-10175.2349
C01603=9.959,70.362,53.146,160.4056,25.5283,-10178.0561
C01604=11.825,72.328,54.436,175.3679,1.0293,-10179.2852
C01605=12.951,75.822,56.240,-177.3643,-0.2478,-10179.6930
C01606=13.963,80.549,58.128,-174.0620,-0.3468,-10179.8344
C01607=15.041,85.905,59.597,-172.0939,-0.5331,-10179.9312
C01608=16.396,90.884,60.330,-172.2930,-2.2395,-10180.2265
C01609=19.672,94.474,60.719,-176.6107,-3.5414,-10181.7624
C01610=24.496,96.092,61.037,-179.1715,-2.3205,-10184.3014
C01611=29.931,95.359,61.359,-179.9991,-0.1559,-10187.4259
C01612=35.488,93.484,61.571,-179.9993,-0.0181,-10190.7876
C01613=41.009,91.197,61.571,-179.9982,-0.0180,-10194.2123
C01614=46.265,88.593,61.359,179.9976,-0.1564,-10197.5744
C01615=50.626,85.269,61.037,179.1730,-2.3238,-10200.6985
C01616=52.893,80.714,60.719,176.6123,-3.5381,-10203.2374
C01617=52.671,75.858,60.330,172.2916,-2.2418,-10204.7737
C01618=50.109,71.379,59.597,172.0924,-0.5334,-10205.0694
C01619=47.084,66.830,58.128,174.0623,-0.3437,-10205.1660
C01620=44.457,62.772,56.240,177.3670,-0.2495,-10205.3073
C01621=42.782,59.505,54.436,-175.3684,1.0288,-10205.7148
C01622=42.712,56.796,53.146,-160.4096,25.5319,-10206.9441
C01623=44.952,54.020,52.637,-175.1533,38.4356,-10209.7651
C01624=47.437,51.781,52.615,179.7155,39.0245,-10212.4931
C01625=49.656,49.656,52.630,179.9948,39.0149,-10215.0000
C01626=51.781,47.437,52.615,-179.7155,39.0245,-10217.5069
C01627=54.020,44.952,52.637,175.1533,38.4356,-10220.2349
C01628=56.796,42.711,53.146,160.4094,25.5317,-10223.0566
C01629=59.505,42.782,54.436,175.3684,1.0288,-10224.2852
C01630=62.772,44.457,56.240,-177.3670,-0.2495,-10224.6927
C01631=66.830,47.084,58.128,-174.0623,-0.3437,-10224.8340
C01632=71.379,50.109,59.597,-172.0924,-0.5334,-10224.9306
C01633=75.858,52.671,60.330,-172.2916,-2.2418,-10225.2263
C01634=80.714,52.893,60.719,-176.6123,-3.5381,-10226.7626
C01635=85.269,50.626,61.037,-179.1730,-2.3238,-10229.3015
C01636=88.593,46.265,61.359,-179.9976,-0.1564,-10232.4256
C01637=91.197,41.009,61.571,179.9982,-0.0180,-10235.7877
C01638=93.484,35.488,61.571,179.9993,-0.0181,-10239.2124
C01639=95.359,29.931,61.359,179.9991,-0.1559,-10242.5741
C01640=96.092,24.496,61.037,179.1715,-2.3205,-10245.6986
C01641=94.474,19.672,60.719,176.6107,-3.5414,-10248.2376
C01642=90.884,16.396,60.330,172.2930,-2.2395,-10249.7735
C01643=85.905,15.041,59.597,172.0939,-0.5331,-10250.0688
C01644=80.549,13.963,58.128,174.0620,-0.3468,-10250.1656
C01645=75.822,12.951,56.240,177.3643,-0.2478,-10250.3070
C01646=72.328,11.825,54.436,-175.3679,1.0293,-10250.7148
C01647=70.362,9.959,53.146,-160.4056,25.5283,-10251.9439
C01648=69.984,6.412,52.637,-175.1539,38.4339,-10254.7651
C01649=70.158,3.072,52.615,179.7154,39.0245,-10257.4928
C01650=70.224,0.000,52.630,180.0000,39.0133,-10260.0000
C01651=70.158,-3.071,52.615,-179.7148,39.0245,-10262.5064
C01652=69.984,-6.412,52.637,175.1539,38.4339,-10265.2349
C01653=70.362,-9.959,53.146,160.4106,25.5345,-10268.0561
C01654=72.328,-11.825,54.436,175.3679,1.0293,-10269.2852
C01655=75.822,-12.951,56.240,-177.3643,-0.2478,-10269.6930
C01656=80.549,-13.963,58.128,-174.0620,-0.3468,-10269.8344
C01657=85.905,-15.041,59.597,-172.0939,-0.5331,-10269.9312
C01658=90.884,-16.396,60.330,-172.2930,-2.2395,-10270.2265
C01659=94.474,-19.672,60.719,-176.6107,-3.5414,-10271.7624
C01660=96.092,-24.496,61.037,-179.1715,-2.3205,-10274.3014
C01661=95.359,-29.931,61.359,-179.9991,-0.1559,-10277.4259
C01662=93.484,-35.488,61.571,-179.9993,-0.0181,-10280.7876
C01663=91.197,-41.009,61.571,-179.9982,-0.0180,-10284.2123
C01664=88.593,-46.265,61.359,179.9976,-0.1564,-10287.5744
C01665=85.269,-50.626,61.037,179.1730,-2.3238,-10290.6985
C01666=80.714,-52.893,60.719,176.6123,-3.5381,-10293.2374
C01667=75.858,-52.671,60.330,172.2916,-2.2418,-10294.7737
C01668=71.379,-50.109,59.597,172.0924,-0.5334,-10295.0694
C01669=66.830,-47.084,58.128,174.0623,-0.3437,-10295.1660
C01670=62.772,-44.457,56.240,177.3670,-0.2495,-10295.3073
C01671=59.505,-42.782,54.436,-175.3684,1.0288,-10295.7148
C01672=56.796,-42.712,53.146,-160.4096,25.5319,-10296.9441
C01673=54.020,-44.952,52.637,-175.1533,38.4356,-10299.7651
C01674=51.781,-47.437,52.615,179.7155,39.0245,-10302.4931
C01675=49.656,-49.656,52.630,179.9948,39.0149,-10305.0000
C01676=47.437,-51.781,52.615,-179.7155,39.0245,-10307.5069
C01677=44.952,-54.020,52.637,175.1533,38.4356,-10310.2349
C01678=42.711,-56.796,53.146,160.4094,25.5317,-10313.0566
C01679=42.782,-59.505,54.436,175.3684,1.0288,-10314.2852
C01680=44.457,-62.772,56.240,-177.3670,-0.2495,-10314.6927
C01681=47.084,-66.830,58.128,-174.0623,-0.3437,-10314.8340
C01682=50.109,-71.379,59.597,-172.0924,-0.5334,-10314.9306
C01683=52.671,-75.858,60.330,-172.2916,-2.2418,-10315.2263
C01684=52.893,-80.714,60.719,-176.6123,-3.5381,-10316.7626
C01685=50.626,-85.269,61.037,-179.1730,-2.3238,-10319.3015
C01686=46.265,-88.593,61.359,-179.9976,-0.1564,-10322.4256
C01687=41.009,-91.197,61.571,179.9982,-0.0180,-10325.7877
C01688=35.488,-93.484,61.571,179.9993,-0.0181,-10329.2124
C01689=29.931,-95.359,61.359,179.9991,-0.1559,-10332.5741
C01690=24.496,-96.092,61.037,179.1715,-2.3205,-10335.6986
C01691=19.672,-94.474,60.719,176.6107,-3.5414,-10338.2376
C01692=16.396,-90.884,60.330,172.2930,-2.2395,-10339.7735
C01693=15.041,-85.905,59.597,172.0939,-0.5331,-10340.0688
C01694=13.963,-80.549,58.128,174.0620,-0.3468,-10340.1656
C01695=12.951,-75.822,56.240,177.3643,-0.2478,-10340.3070
C01696=11.825,-72.328,54.436,-175.3679,1.0293,-10340.7148
C01697=9.959,-70.362,53.146,-160.4056,25.5283,-10341.9439
C01698=6.412,-69.984,52.637,-175.1539,38.4339,-10344.7651
C01699=3.072,-70.158,52.615,179.7154,39.0245,-10347.4928
C01700=0.000,-70.224,52.630,180.0000,39.0133,-10350.0000
C01701=-3.071,-70.158,52.615,-179.7148,39.0245,-10352.5064
C01702=-6.412,-69.984,52.637,175.1539,38.4339,-10355.2349
C01703=-9.959,-70.362,53.146,160.4106,25.5345,-10358.0561
C01704=-11.825,-72.328,54.436,175.3679,1.0293,-10359.2852
C01705=-12.951,-75.822,56.240,-177.3643,-0.2478,-10359.6930
C01706=-13.963,-80.549,58.128,-174.0620,-0.3468,-10359.8344
C01707=-15.041,-85.905,59.597,-172.0939,-0.5331,-10359.9312
C01708=-16.396,-90.884,60.330,-172.2930,-2.2395,-10360.2265
C01709=-19.672,-94.474,60.719,-176.6107,-3.5414,-10361.7624
C01710=-24.496,-96.092,61.037,-179.1715,-2.3205,-10364.3014
C01711=-29.931,-95.359,61.359,-179.9991,-0.1559,-10367.4259
C01712=-35.488,-93.484,61.571,-179.9993,-0.0181,-10370.7876
C01713=-41.009,-91.197,61.571,-179.9982,-0.0180,-10374.2123
C01714=-46.265,-88.593,61.359,179.9976,-0.1564,-10377.5744
C01715=-50.626,-85.269,61.037,179.1730,-2.3238,-10380.6985
C01716=-52.893,-80.714,60.719,176.6123,-3.5381,-10383.2374
C01717=-52.671,-75.858,60.330,172.2916,-2.2418,-10384.7737
C01718=-50.109,-71.379,59.597,172.0924,-0.5334,-10385.0694
C01719=-47.084,-66.830,58.128,174.0623,-0.3437,-10385.1660
C01720=-44.457,-62.772,56.240,177.3670,-0.2495,-10385.3073
C01721=-42.782,-59.505,54.436,-175.3684,1.0288,-10385.7148
C01722=-42.712,-56.796,53.146,-160.4096,25.5319,-10386.9441
C01723=-44.952,-54.020,52.637,-175.1533,38.4356,-10389.7651
C01724=-47.437,-51.781,52.615,179.7155,39.0245,-10392.4931
C01725=-49.656,-49.656,52.630,179.9948,39.0149,-10395.0000
C01726=-51.781,-47.437,52.615,-179.7155,39.0245,-10397.5069
C01727=-54.020,-44.952,52.637,175.1533,38.4356,-10400.2349
C01728=-56.796,-42.711,53.146,160.4094,25.5317,-10403.0566
C01729=-59.505,-42.782,54.436,175.3684,1.0288,-10404.2852
C01730=-62.772,-44.457,56.240,-177.3670,-0.2495,-10404.6927
C01731=-66.830,-47.084,58.128,-174.0623,-0.3437,-10404.8340
C01732=-71.379,-50.109,59.597,-172.0924,-0.5334,-10404.9306
C01733=-75.858,-52.671,60.330,-172.2916,-2.2418,-10405.2263
C01734=-80.714,-52.893,60.719,-176.6123,-3.5381,-10406.7626
